(* IEC 61131-3 sources: UniTest/iecUnitTest_br/Global, 102 files *)

(* ---- Global.typ ---- *)
TYPE
    utTestCase :    STRUCT
        id : UINT; (*Identifier of the test*)
        desc : ARRAY[0..4] OF STRING[255]; (*Description of the test case*)
        state : utTestCaseStates; (*State of the test*)
        msg : STRING[255]; (*Result of the test*)
    END_STRUCT;
    utTestCaseStates :
    (
        SETUP := 0, (**)
        RUNNING := 1, (**)
        PASSED := 2, (**)
        FAILED := 3, (**)
    )
    utTestCaseSummary :    STRUCT
        Id : UINT; (*Id of the test object. Must be unique number*)
        Name : STRING[250]; (*Name of the test object*)
        TotalTests : UINT; (*Total number of tests existing*)
        TestsPassed : UINT; (*Number of tests passed*)
        TestsFailed : UINT; (*Number of tests failed*)
        PassRate : REAL; (*Pass rate % of the tests*)
        TestsRunning : BOOL; (*One or more tests are running*)
        Error : utErrors; (*Error code if error occured*)
    END_STRUCT;
    utErrors :
    (
        NO_ERROR := 0, (**)
        NO_TEST_CASES_DEFINED := 100, (**)
    )
END_TYPE

(* ---- assertArrayEqual_BYTE.st ---- *)
FUNCTION assertArrayEqual_BYTE
    (*https://github.com/tkucic/iecUnitTest/blob/main/docs/docs/ns/Global/fc/assertArrayEqual_BYTE.md*)
    vStop := (size / SIZEOF(act^[0])) - 1;

    FOR i:=0 TO vStop DO
    	pt1 := ADR(act^[i]);
    	pt2 := ADR(xp^[i]);
    	IF pt1^ <> pt2^ THEN
    		assertArrayEqual_BYTE := FALSE;
    		RETURN;
    	END_IF
    END_FOR
    (*If we reach here, all elements are equal*)
    assertArrayEqual_BYTE := TRUE;
    RETURN;

END_FUNCTION

(* ---- assertArrayEqual_DINT.st ---- *)
FUNCTION assertArrayEqual_DINT
    (*https://github.com/tkucic/iecUnitTest/blob/main/docs/docs/ns/Global/fc/assertArrayEqual_DINT.md*)
    vStop := (size / SIZEOF(act^[0])) - 1;

    FOR i:=0 TO vStop DO
    	pt1 := ADR(act^[i]);
    	pt2 := ADR(xp^[i]);
    	IF pt1^ <> pt2^ THEN
    		assertArrayEqual_DINT := FALSE;
    		RETURN;
    	END_IF
    END_FOR
    (*If we reach here, all elements are equal*)
    assertArrayEqual_DINT := TRUE;
    RETURN;

END_FUNCTION

(* ---- assertArrayEqual_DWORD.st ---- *)
FUNCTION assertArrayEqual_DWORD
    (*https://github.com/tkucic/iecUnitTest/blob/main/docs/docs/ns/Global/fc/assertArrayEqual_DWORD.md*)
    vStop := (size / SIZEOF(act^[0])) - 1;

    FOR i:=0 TO vStop DO
    	pt1 := ADR(act^[i]);
    	pt2 := ADR(xp^[i]);
    	IF pt1^ <> pt2^ THEN
    		assertArrayEqual_DWORD := FALSE;
    		RETURN;
    	END_IF
    END_FOR
    (*If we reach here, all elements are equal*)
    assertArrayEqual_DWORD := TRUE;
    RETURN;

END_FUNCTION

(* ---- assertArrayEqual_INT.st ---- *)
FUNCTION assertArrayEqual_INT
    (*https://github.com/tkucic/iecUnitTest/blob/main/docs/docs/ns/Global/fc/assertArrayEqual_INT.md*)
    vStop := (size / SIZEOF(act^[0])) - 1;

    FOR i:=0 TO vStop DO
    	pt1 := ADR(act^[i]);
    	pt2 := ADR(xp^[i]);
    	IF pt1^ <> pt2^ THEN
    		assertArrayEqual_INT := FALSE;
    		RETURN;
    	END_IF
    END_FOR
    (*If we reach here, all elements are equal*)
    assertArrayEqual_INT := TRUE;
    RETURN;

END_FUNCTION

(* ---- assertArrayEqual_LDATE.st ---- *)
FUNCTION assertArrayEqual_LDATE
    (*https://github.com/tkucic/iecUnitTest/blob/main/docs/docs/ns/Global/fc/assertArrayEqual_LDATE.md*)
    vStop := (size / SIZEOF(act^[0])) - 1;

    FOR i:=0 TO vStop DO
    	pt1 := ADR(act^[i]);
    	pt2 := ADR(xp^[i]);
    	IF pt1^ <> pt2^ THEN
    		assertArrayEqual_LDATE := FALSE;
    		RETURN;
    	END_IF
    END_FOR
    (*If we reach here, all elements are equal*)
    assertArrayEqual_LDATE := TRUE;
    RETURN;

END_FUNCTION

(* ---- assertArrayEqual_LINT.st ---- *)
FUNCTION assertArrayEqual_LINT
    (*https://github.com/tkucic/iecUnitTest/blob/main/docs/docs/ns/Global/fc/assertArrayEqual_LINT.md*)
    vStop := (size / SIZEOF(act^[0])) - 1;

    FOR i:=0 TO vStop DO
    	pt1 := ADR(act^[i]);
    	pt2 := ADR(xp^[i]);
    	IF pt1^ <> pt2^ THEN
    		assertArrayEqual_LINT := FALSE;
    		RETURN;
    	END_IF
    END_FOR
    (*If we reach here, all elements are equal*)
    assertArrayEqual_LINT := TRUE;
    RETURN;

END_FUNCTION

(* ---- assertArrayEqual_LREAL.st ---- *)
FUNCTION assertArrayEqual_LREAL
    (*https://github.com/tkucic/iecUnitTest/blob/main/docs/docs/ns/Global/fc/assertArrayEqual_LREAL.md*)
    vStop := (size / SIZEOF(act^[0])) - 1;

    FOR i:=0 TO vStop DO
    	pt1 := ADR(act^[i]);
    	pt2 := ADR(xp^[i]);
    	IF pt1^ <> pt2^ THEN
    		assertArrayEqual_LREAL := FALSE;
    		RETURN;
    	END_IF
    END_FOR
    (*If we reach here, all elements are equal*)
    assertArrayEqual_LREAL := TRUE;
    RETURN;

END_FUNCTION

(* ---- assertArrayEqual_LTIME_OF_DAY.st ---- *)
FUNCTION assertArrayEqual_LTIME_OF_DAY
    (*https://github.com/tkucic/iecUnitTest/blob/main/docs/docs/ns/Global/fc/assertArrayEqual_LTIME_OF_DAY.md*)
    vStop := (size / SIZEOF(act^[0])) - 1;

    FOR i:=0 TO vStop DO
    	pt1 := ADR(act^[i]);
    	pt2 := ADR(xp^[i]);
    	IF pt1^ <> pt2^ THEN
    		assertArrayEqual_LTIME_OF_DAY := FALSE;
    		RETURN;
    	END_IF
    END_FOR
    (*If we reach here, all elements are equal*)
    assertArrayEqual_LTIME_OF_DAY := TRUE;
    RETURN;

END_FUNCTION

(* ---- assertArrayEqual_LWORD.st ---- *)
FUNCTION assertArrayEqual_LWORD
    (*https://github.com/tkucic/iecUnitTest/blob/main/docs/docs/ns/Global/fc/assertArrayEqual_LWORD.md*)
    vStop := (size / SIZEOF(act^[0])) - 1;

    FOR i:=0 TO vStop DO
    	pt1 := ADR(act^[i]);
    	pt2 := ADR(xp^[i]);
    	IF pt1^ <> pt2^ THEN
    		assertArrayEqual_LWORD := FALSE;
    		RETURN;
    	END_IF
    END_FOR
    (*If we reach here, all elements are equal*)
    assertArrayEqual_LWORD := TRUE;
    RETURN;

END_FUNCTION

(* ---- assertArrayEqual_SINT.st ---- *)
FUNCTION assertArrayEqual_SINT
    (*https://github.com/tkucic/iecUnitTest/blob/main/docs/docs/ns/Global/fc/assertArrayEqual_SINT.md*)
    vStop := (size / SIZEOF(act^[0])) - 1;

    FOR i:=0 TO vStop DO
    	pt1 := ADR(act^[i]);
    	pt2 := ADR(xp^[i]);
    	IF pt1^ <> pt2^ THEN
    		assertArrayEqual_SINT := FALSE;
    		RETURN;
    	END_IF
    END_FOR
    (*If we reach here, all elements are equal*)
    assertArrayEqual_SINT := TRUE;
    RETURN;

END_FUNCTION

(* ---- assertArrayEqual_STRING.st ---- *)
FUNCTION assertArrayEqual_STRING
    (*https://github.com/tkucic/iecUnitTest/blob/main/docs/docs/ns/Global/fc/assertArrayEqual_STRING.md*)
    vStop := (size / SIZEOF(act^[0])) - 1;

    FOR i:=0 TO vStop DO
    	pt1 := ADR(act^[i]);
    	pt2 := ADR(xp^[i]);
    	IF pt1^ <> pt2^ THEN
    		assertArrayEqual_STRING := FALSE;
    		RETURN;
    	END_IF
    END_FOR
    (*If we reach here, all elements are equal*)
    assertArrayEqual_STRING := TRUE;
    RETURN;

END_FUNCTION

(* ---- assertArrayEqual_TIME.st ---- *)
FUNCTION assertArrayEqual_TIME
    (*https://github.com/tkucic/iecUnitTest/blob/main/docs/docs/ns/Global/fc/assertArrayEqual_TIME.md*)
    vStop := (size / SIZEOF(act^[0])) - 1;

    FOR i:=0 TO vStop DO
    	pt1 := ADR(act^[i]);
    	pt2 := ADR(xp^[i]);
    	IF pt1^ <> pt2^ THEN
    		assertArrayEqual_TIME := FALSE;
    		RETURN;
    	END_IF
    END_FOR
    (*If we reach here, all elements are equal*)
    assertArrayEqual_TIME := TRUE;
    RETURN;

END_FUNCTION

(* ---- assertArrayEqual_UDINT.st ---- *)
FUNCTION assertArrayEqual_UDINT
    (*https://github.com/tkucic/iecUnitTest/blob/main/docs/docs/ns/Global/fc/assertArrayEqual_UDINT.md*)
    vStop := (size / SIZEOF(act^[0])) - 1;

    FOR i:=0 TO vStop DO
    	pt1 := ADR(act^[i]);
    	pt2 := ADR(xp^[i]);
    	IF pt1^ <> pt2^ THEN
    		assertArrayEqual_UDINT := FALSE;
    		RETURN;
    	END_IF
    END_FOR
    (*If we reach here, all elements are equal*)
    assertArrayEqual_UDINT := TRUE;
    RETURN;

END_FUNCTION

(* ---- assertArrayEqual_UINT.st ---- *)
FUNCTION assertArrayEqual_UINT
    (*https://github.com/tkucic/iecUnitTest/blob/main/docs/docs/ns/Global/fc/assertArrayEqual_UINT.md*)
    vStop := (size / SIZEOF(act^[0])) - 1;

    FOR i:=0 TO vStop DO
    	pt1 := ADR(act^[i]);
    	pt2 := ADR(xp^[i]);
    	IF pt1^ <> pt2^ THEN
    		assertArrayEqual_UINT := FALSE;
    		RETURN;
    	END_IF
    END_FOR
    (*If we reach here, all elements are equal*)
    assertArrayEqual_UINT := TRUE;
    RETURN;

END_FUNCTION

(* ---- assertArrayEqual_ULINT.st ---- *)
FUNCTION assertArrayEqual_ULINT
    (*https://github.com/tkucic/iecUnitTest/blob/main/docs/docs/ns/Global/fc/assertArrayEqual_ULINT.md*)
    vStop := (size / SIZEOF(act^[0])) - 1;

    FOR i:=0 TO vStop DO
    	pt1 := ADR(act^[i]);
    	pt2 := ADR(xp^[i]);
    	IF pt1^ <> pt2^ THEN
    		assertArrayEqual_ULINT := FALSE;
    		RETURN;
    	END_IF
    END_FOR
    (*If we reach here, all elements are equal*)
    assertArrayEqual_ULINT := TRUE;
    RETURN;

END_FUNCTION

(* ---- assertArrayEqual_WORD.st ---- *)
FUNCTION assertArrayEqual_WORD
    (*https://github.com/tkucic/iecUnitTest/blob/main/docs/docs/ns/Global/fc/assertArrayEqual_WORD.md*)
    vStop := (size / SIZEOF(act^[0])) - 1;

    FOR i:=0 TO vStop DO
    	pt1 := ADR(act^[i]);
    	pt2 := ADR(xp^[i]);
    	IF pt1^ <> pt2^ THEN
    		assertArrayEqual_WORD := FALSE;
    		RETURN;
    	END_IF
    END_FOR
    (*If we reach here, all elements are equal*)
    assertArrayEqual_WORD := TRUE;
    RETURN;

END_FUNCTION

(* ---- assertArrayEqual_WSTRING.st ---- *)
FUNCTION assertArrayEqual_WSTRING
    (*https://github.com/tkucic/iecUnitTest/blob/main/docs/docs/ns/Global/fc/assertArrayEqual_WSTRING.md*)
    vStop := (size / SIZEOF(act^[0])) - 1;

    FOR i:=0 TO vStop DO
    	pt1 := ADR(act^[i]);
    	pt2 := ADR(xp^[i]);
    	IF pt1^ <> pt2^ THEN
    		assertArrayEqual_WSTRING := FALSE;
    		RETURN;
    	END_IF
    END_FOR
    (*If we reach here, all elements are equal*)
    assertArrayEqual_WSTRING := TRUE;
    RETURN;

END_FUNCTION

(* ---- assertEqual_BYTE.st ---- *)
FUNCTION assertEqual_BYTE
    (*https://github.com/tkucic/iecUnitTest/blob/main/docs/docs/ns/Global/fc/assertEqual_BYTE.md*)
    assertEqual_BYTE := act = xp;
    RETURN;

END_FUNCTION

(* ---- assertEqual_DATE_AND_TIME.st ---- *)
FUNCTION assertEqual_DATE_AND_TIME
    (*https://github.com/tkucic/iecUnitTest/blob/main/docs/docs/ns/Global/fc/assertEqual_DATE_AND_TIME.md*)
    assertEqual_DATE_AND_TIME := act = xp;
    RETURN;

END_FUNCTION

(* ---- assertEqual_DWORD.st ---- *)
FUNCTION assertEqual_DWORD
    (*https://github.com/tkucic/iecUnitTest/blob/main/docs/docs/ns/Global/fc/assertEqual_DWORD.md*)
    assertEqual_DWORD := act = xp;
    RETURN;

END_FUNCTION

(* ---- assertEqual_INT.st ---- *)
FUNCTION assertEqual_INT
    (*https://github.com/tkucic/iecUnitTest/blob/main/docs/docs/ns/Global/fc/assertEqual_INT.md*)
    assertEqual_INT := act = xp;
    RETURN;

END_FUNCTION

(* ---- assertEqual_LDATE.st ---- *)
FUNCTION assertEqual_LDATE
    (*https://github.com/tkucic/iecUnitTest/blob/main/docs/docs/ns/Global/fc/assertEqual_LDATE.md*)
    assertEqual_LDATE := act = xp;
    RETURN;

END_FUNCTION

(* ---- assertEqual_LDATE_AND_TIME.st ---- *)
FUNCTION assertEqual_LDATE_AND_TIME
    (*https://github.com/tkucic/iecUnitTest/blob/main/docs/docs/ns/Global/fc/assertEqual_LDATE_AND_TIME.md*)
    assertEqual_LDATE_AND_TIME := act = xp;
    RETURN;

END_FUNCTION

(* ---- assertEqual_LINT.st ---- *)
FUNCTION assertEqual_LINT
    (*https://github.com/tkucic/iecUnitTest/blob/main/docs/docs/ns/Global/fc/assertEqual_LINT.md*)
    assertEqual_LINT := act = xp;
    RETURN;

END_FUNCTION

(* ---- assertEqual_LTIME.st ---- *)
FUNCTION assertEqual_LTIME
    (*https://github.com/tkucic/iecUnitTest/blob/main/docs/docs/ns/Global/fc/assertEqual_LTIME.md*)
    assertEqual_LTIME := act = xp;
    RETURN;

END_FUNCTION

(* ---- assertEqual_LTIME_OF_DAY.st ---- *)
FUNCTION assertEqual_LTIME_OF_DAY
    (*https://github.com/tkucic/iecUnitTest/blob/main/docs/docs/ns/Global/fc/assertEqual_LTIME_OF_DAY.md*)
    assertEqual_LTIME_OF_DAY := act = xp;
    RETURN;

END_FUNCTION

(* ---- assertEqual_REAL.st ---- *)
FUNCTION assertEqual_REAL
    (*https://github.com/tkucic/iecUnitTest/blob/main/docs/docs/ns/Global/fc/assertEqual_REAL.md*)
    assertEqual_REAL := act = xp;
    RETURN;

END_FUNCTION

(* ---- assertEqual_STRING.st ---- *)
FUNCTION assertEqual_STRING
    (*https://github.com/tkucic/iecUnitTest/blob/main/docs/docs/ns/Global/fc/assertEqual_STRING.md*)
    assertEqual_STRING := act = xp;
    RETURN;

END_FUNCTION

(* ---- assertEqual_UDINT.st ---- *)
FUNCTION assertEqual_UDINT
    (*https://github.com/tkucic/iecUnitTest/blob/main/docs/docs/ns/Global/fc/assertEqual_UDINT.md*)
    assertEqual_UDINT := act = xp;
    RETURN;

END_FUNCTION

(* ---- assertEqual_ULINT.st ---- *)
FUNCTION assertEqual_ULINT
    (*https://github.com/tkucic/iecUnitTest/blob/main/docs/docs/ns/Global/fc/assertEqual_ULINT.md*)
    assertEqual_ULINT := act = xp;
    RETURN;

END_FUNCTION

(* ---- assertEqual_USINT.st ---- *)
FUNCTION assertEqual_USINT
    (*https://github.com/tkucic/iecUnitTest/blob/main/docs/docs/ns/Global/fc/assertEqual_USINT.md*)
    assertEqual_USINT := act = xp;
    RETURN;

END_FUNCTION

(* ---- assertFalse.st ---- *)
FUNCTION assertFalse
    (*https://github.com/tkucic/iecUnitTest/blob/main/docs/docs/ns/Global/fc/assertFalse.md*)
    assertFalse := NOT condition;
    RETURN;

END_FUNCTION

(* ---- assertGreater_BYTE.st ---- *)
FUNCTION assertGreater_BYTE
    (*https://github.com/tkucic/iecUnitTest/blob/main/docs/docs/ns/Global/fc/assertGreater_BYTE.md*)
    assertGreater_BYTE := act > xp;
    RETURN;

END_FUNCTION

(* ---- assertGreater_DATE.st ---- *)
FUNCTION assertGreater_DATE
    (*https://github.com/tkucic/iecUnitTest/blob/main/docs/docs/ns/Global/fc/assertGreater_DATE.md*)
    assertGreater_DATE := act > xp;
    RETURN;

END_FUNCTION

(* ---- assertGreater_DWORD.st ---- *)
FUNCTION assertGreater_DWORD
    (*https://github.com/tkucic/iecUnitTest/blob/main/docs/docs/ns/Global/fc/assertGreater_DWORD.md*)
    assertGreater_DWORD := act > xp;
    RETURN;

END_FUNCTION

(* ---- assertGreater_INT.st ---- *)
FUNCTION assertGreater_INT
    (*https://github.com/tkucic/iecUnitTest/blob/main/docs/docs/ns/Global/fc/assertGreater_INT.md*)
    assertGreater_INT := act > xp;
    RETURN;

END_FUNCTION

(* ---- assertGreater_LDATE_AND_TIME.st ---- *)
FUNCTION assertGreater_LDATE_AND_TIME
    (*https://github.com/tkucic/iecUnitTest/blob/main/docs/docs/ns/Global/fc/assertGreater_LDATE_AND_TIME.md*)
    assertGreater_LDATE_AND_TIME := act > xp;
    RETURN;

END_FUNCTION

(* ---- assertGreater_LREAL.st ---- *)
FUNCTION assertGreater_LREAL
    (*https://github.com/tkucic/iecUnitTest/blob/main/docs/docs/ns/Global/fc/assertGreater_LREAL.md*)
    assertGreater_LREAL := act > xp;
    RETURN;

END_FUNCTION

(* ---- assertGreater_LTIME.st ---- *)
FUNCTION assertGreater_LTIME
    (*https://github.com/tkucic/iecUnitTest/blob/main/docs/docs/ns/Global/fc/assertGreater_LTIME.md*)
    assertGreater_LTIME := act > xp;
    RETURN;

END_FUNCTION

(* ---- assertGreater_LTIME_OF_DAY.st ---- *)
FUNCTION assertGreater_LTIME_OF_DAY
    (*https://github.com/tkucic/iecUnitTest/blob/main/docs/docs/ns/Global/fc/assertGreater_LTIME_OF_DAY.md*)
    assertGreater_LTIME_OF_DAY := act > xp;
    RETURN;

END_FUNCTION

(* ---- assertGreater_LWORD.st ---- *)
FUNCTION assertGreater_LWORD
    (*https://github.com/tkucic/iecUnitTest/blob/main/docs/docs/ns/Global/fc/assertGreater_LWORD.md*)
    assertGreater_LWORD := act > xp;
    RETURN;

END_FUNCTION

(* ---- assertGreater_REAL.st ---- *)
FUNCTION assertGreater_REAL
    (*https://github.com/tkucic/iecUnitTest/blob/main/docs/docs/ns/Global/fc/assertGreater_REAL.md*)
    assertGreater_REAL := act > xp;
    RETURN;

END_FUNCTION

(* ---- assertGreater_SINT.st ---- *)
FUNCTION assertGreater_SINT
    (*https://github.com/tkucic/iecUnitTest/blob/main/docs/docs/ns/Global/fc/assertGreater_SINT.md*)
    assertGreater_SINT := act > xp;
    RETURN;

END_FUNCTION

(* ---- assertGreater_TIME.st ---- *)
FUNCTION assertGreater_TIME
    (*https://github.com/tkucic/iecUnitTest/blob/main/docs/docs/ns/Global/fc/assertGreater_TIME.md*)
    assertGreater_TIME := act > xp;
    RETURN;

END_FUNCTION

(* ---- assertGreater_TIME_OF_DAY.st ---- *)
FUNCTION assertGreater_TIME_OF_DAY
    (*https://github.com/tkucic/iecUnitTest/blob/main/docs/docs/ns/Global/fc/assertGreater_TIME_OF_DAY.md*)
    assertGreater_TIME_OF_DAY := act > xp;
    RETURN;

END_FUNCTION

(* ---- assertGreater_UINT.st ---- *)
FUNCTION assertGreater_UINT
    (*https://github.com/tkucic/iecUnitTest/blob/main/docs/docs/ns/Global/fc/assertGreater_UINT.md*)
    assertGreater_UINT := act > xp;
    RETURN;

END_FUNCTION

(* ---- assertGreater_ULINT.st ---- *)
FUNCTION assertGreater_ULINT
    (*https://github.com/tkucic/iecUnitTest/blob/main/docs/docs/ns/Global/fc/assertGreater_ULINT.md*)
    assertGreater_ULINT := act > xp;
    RETURN;

END_FUNCTION

(* ---- assertGreater_WORD.st ---- *)
FUNCTION assertGreater_WORD
    (*https://github.com/tkucic/iecUnitTest/blob/main/docs/docs/ns/Global/fc/assertGreater_WORD.md*)
    assertGreater_WORD := act > xp;
    RETURN;

END_FUNCTION

(* ---- assertGreaterEqual_BYTE.st ---- *)
FUNCTION assertGreaterEqual_BYTE
    (*https://github.com/tkucic/iecUnitTest/blob/main/docs/docs/ns/Global/fc/assertGreaterEqual_BYTE.md*)
    assertGreaterEqual_BYTE := act >= xp;
    RETURN;

END_FUNCTION

(* ---- assertGreaterEqual_DWORD.st ---- *)
FUNCTION assertGreaterEqual_DWORD
    (*https://github.com/tkucic/iecUnitTest/blob/main/docs/docs/ns/Global/fc/assertGreaterEqual_DWORD.md*)
    assertGreaterEqual_DWORD := act >= xp;
    RETURN;

END_FUNCTION

(* ---- assertGreaterEqual_LDATE_AND_TIME.st ---- *)
FUNCTION assertGreaterEqual_LDATE_AND_TIME
    (*https://github.com/tkucic/iecUnitTest/blob/main/docs/docs/ns/Global/fc/assertGreaterEqual_LDATE_AND_TIME.md*)
    assertGreaterEqual_LDATE_AND_TIME := act >= xp;
    RETURN;

END_FUNCTION

(* ---- assertGreaterEqual_LTIME_OF_DAY.st ---- *)
FUNCTION assertGreaterEqual_LTIME_OF_DAY
    (*https://github.com/tkucic/iecUnitTest/blob/main/docs/docs/ns/Global/fc/assertGreaterEqual_LTIME_OF_DAY.md*)
    assertGreaterEqual_LTIME_OF_DAY := act >= xp;
    RETURN;

END_FUNCTION

(* ---- assertGreaterEqual_LWORD.st ---- *)
FUNCTION assertGreaterEqual_LWORD
    (*https://github.com/tkucic/iecUnitTest/blob/main/docs/docs/ns/Global/fc/assertGreaterEqual_LWORD.md*)
    assertGreaterEqual_LWORD := act >= xp;
    RETURN;

END_FUNCTION

(* ---- assertGreaterEqual_SINT.st ---- *)
FUNCTION assertGreaterEqual_SINT
    (*https://github.com/tkucic/iecUnitTest/blob/main/docs/docs/ns/Global/fc/assertGreaterEqual_SINT.md*)
    assertGreaterEqual_SINT := act >= xp;
    RETURN;

END_FUNCTION

(* ---- assertGreaterEqual_TIME_OF_DAY.st ---- *)
FUNCTION assertGreaterEqual_TIME_OF_DAY
    (*https://github.com/tkucic/iecUnitTest/blob/main/docs/docs/ns/Global/fc/assertGreaterEqual_TIME_OF_DAY.md*)
    assertGreaterEqual_TIME_OF_DAY := act >= xp;
    RETURN;

END_FUNCTION

(* ---- assertGreaterEqual_UDINT.st ---- *)
FUNCTION assertGreaterEqual_UDINT
    (*https://github.com/tkucic/iecUnitTest/blob/main/docs/docs/ns/Global/fc/assertGreaterEqual_UDINT.md*)
    assertGreaterEqual_UDINT := act >= xp;
    RETURN;

END_FUNCTION

(* ---- assertGreaterEqual_UINT.st ---- *)
FUNCTION assertGreaterEqual_UINT
    (*https://github.com/tkucic/iecUnitTest/blob/main/docs/docs/ns/Global/fc/assertGreaterEqual_UINT.md*)
    assertGreaterEqual_UINT := act >= xp;
    RETURN;

END_FUNCTION

(* ---- assertGreaterEqual_ULINT.st ---- *)
FUNCTION assertGreaterEqual_ULINT
    (*https://github.com/tkucic/iecUnitTest/blob/main/docs/docs/ns/Global/fc/assertGreaterEqual_ULINT.md*)
    assertGreaterEqual_ULINT := act >= xp;
    RETURN;

END_FUNCTION

(* ---- assertGreaterEqual_USINT.st ---- *)
FUNCTION assertGreaterEqual_USINT
    (*https://github.com/tkucic/iecUnitTest/blob/main/docs/docs/ns/Global/fc/assertGreaterEqual_USINT.md*)
    assertGreaterEqual_USINT := act >= xp;
    RETURN;

END_FUNCTION

(* ---- assertLess_DATE_AND_TIME.st ---- *)
FUNCTION assertLess_DATE_AND_TIME
    (*https://github.com/tkucic/iecUnitTest/blob/main/docs/docs/ns/Global/fc/assertLess_DATE_AND_TIME.md*)
    assertLess_DATE_AND_TIME := act < xp;
    RETURN;

END_FUNCTION

(* ---- assertLess_DWORD.st ---- *)
FUNCTION assertLess_DWORD
    (*https://github.com/tkucic/iecUnitTest/blob/main/docs/docs/ns/Global/fc/assertLess_DWORD.md*)
    assertLess_DWORD := act < xp;
    RETURN;

END_FUNCTION

(* ---- assertLess_INT.st ---- *)
FUNCTION assertLess_INT
    (*https://github.com/tkucic/iecUnitTest/blob/main/docs/docs/ns/Global/fc/assertLess_INT.md*)
    assertLess_INT := act < xp;
    RETURN;

END_FUNCTION

(* ---- assertLess_LINT.st ---- *)
FUNCTION assertLess_LINT
    (*https://github.com/tkucic/iecUnitTest/blob/main/docs/docs/ns/Global/fc/assertLess_LINT.md*)
    assertLess_LINT := act < xp;
    RETURN;

END_FUNCTION

(* ---- assertLess_LTIME.st ---- *)
FUNCTION assertLess_LTIME
    (*https://github.com/tkucic/iecUnitTest/blob/main/docs/docs/ns/Global/fc/assertLess_LTIME.md*)
    assertLess_LTIME := act < xp;
    RETURN;

END_FUNCTION

(* ---- assertLess_LTIME_OF_DAY.st ---- *)
FUNCTION assertLess_LTIME_OF_DAY
    (*https://github.com/tkucic/iecUnitTest/blob/main/docs/docs/ns/Global/fc/assertLess_LTIME_OF_DAY.md*)
    assertLess_LTIME_OF_DAY := act < xp;
    RETURN;

END_FUNCTION

(* ---- assertLess_LWORD.st ---- *)
FUNCTION assertLess_LWORD
    (*https://github.com/tkucic/iecUnitTest/blob/main/docs/docs/ns/Global/fc/assertLess_LWORD.md*)
    assertLess_LWORD := act < xp;
    RETURN;

END_FUNCTION

(* ---- assertLess_SINT.st ---- *)
FUNCTION assertLess_SINT
    (*https://github.com/tkucic/iecUnitTest/blob/main/docs/docs/ns/Global/fc/assertLess_SINT.md*)
    assertLess_SINT := act < xp;
    RETURN;

END_FUNCTION

(* ---- assertLess_TIME.st ---- *)
FUNCTION assertLess_TIME
    (*https://github.com/tkucic/iecUnitTest/blob/main/docs/docs/ns/Global/fc/assertLess_TIME.md*)
    assertLess_TIME := act < xp;
    RETURN;

END_FUNCTION

(* ---- assertLess_TIME_OF_DAY.st ---- *)
FUNCTION assertLess_TIME_OF_DAY
    (*https://github.com/tkucic/iecUnitTest/blob/main/docs/docs/ns/Global/fc/assertLess_TIME_OF_DAY.md*)
    assertLess_TIME_OF_DAY := act < xp;
    RETURN;

END_FUNCTION

(* ---- assertLess_UDINT.st ---- *)
FUNCTION assertLess_UDINT
    (*https://github.com/tkucic/iecUnitTest/blob/main/docs/docs/ns/Global/fc/assertLess_UDINT.md*)
    assertLess_UDINT := act < xp;
    RETURN;

END_FUNCTION

(* ---- assertLess_USINT.st ---- *)
FUNCTION assertLess_USINT
    (*https://github.com/tkucic/iecUnitTest/blob/main/docs/docs/ns/Global/fc/assertLess_USINT.md*)
    assertLess_USINT := act < xp;
    RETURN;

END_FUNCTION

(* ---- assertLess_WORD.st ---- *)
FUNCTION assertLess_WORD
    (*https://github.com/tkucic/iecUnitTest/blob/main/docs/docs/ns/Global/fc/assertLess_WORD.md*)
    assertLess_WORD := act < xp;
    RETURN;

END_FUNCTION

(* ---- assertLessEqual_BYTE.st ---- *)
FUNCTION assertLessEqual_BYTE
    (*https://github.com/tkucic/iecUnitTest/blob/main/docs/docs/ns/Global/fc/assertLessEqual_BYTE.md*)
    assertLessEqual_BYTE := act <= xp;
    RETURN;

END_FUNCTION

(* ---- assertLessEqual_DATE.st ---- *)
FUNCTION assertLessEqual_DATE
    (*https://github.com/tkucic/iecUnitTest/blob/main/docs/docs/ns/Global/fc/assertLessEqual_DATE.md*)
    assertLessEqual_DATE := act <= xp;
    RETURN;

END_FUNCTION

(* ---- assertLessEqual_DINT.st ---- *)
FUNCTION assertLessEqual_DINT
    (*https://github.com/tkucic/iecUnitTest/blob/main/docs/docs/ns/Global/fc/assertLessEqual_DINT.md*)
    assertLessEqual_DINT := act <= xp;
    RETURN;

END_FUNCTION

(* ---- assertLessEqual_LDATE.st ---- *)
FUNCTION assertLessEqual_LDATE
    (*https://github.com/tkucic/iecUnitTest/blob/main/docs/docs/ns/Global/fc/assertLessEqual_LDATE.md*)
    assertLessEqual_LDATE := act <= xp;
    RETURN;

END_FUNCTION

(* ---- assertLessEqual_LDATE_AND_TIME.st ---- *)
FUNCTION assertLessEqual_LDATE_AND_TIME
    (*https://github.com/tkucic/iecUnitTest/blob/main/docs/docs/ns/Global/fc/assertLessEqual_LDATE_AND_TIME.md*)
    assertLessEqual_LDATE_AND_TIME := act <= xp;
    RETURN;

END_FUNCTION

(* ---- assertLessEqual_LREAL.st ---- *)
FUNCTION assertLessEqual_LREAL
    (*https://github.com/tkucic/iecUnitTest/blob/main/docs/docs/ns/Global/fc/assertLessEqual_LREAL.md*)
    assertLessEqual_LREAL := act <= xp;
    RETURN;

END_FUNCTION

(* ---- assertLessEqual_LTIME.st ---- *)
FUNCTION assertLessEqual_LTIME
    (*https://github.com/tkucic/iecUnitTest/blob/main/docs/docs/ns/Global/fc/assertLessEqual_LTIME.md*)
    assertLessEqual_LTIME := act <= xp;
    RETURN;

END_FUNCTION

(* ---- assertLessEqual_LTIME_OF_DAY.st ---- *)
FUNCTION assertLessEqual_LTIME_OF_DAY
    (*https://github.com/tkucic/iecUnitTest/blob/main/docs/docs/ns/Global/fc/assertLessEqual_LTIME_OF_DAY.md*)
    assertLessEqual_LTIME_OF_DAY := act <= xp;
    RETURN;

END_FUNCTION

(* ---- assertLessEqual_REAL.st ---- *)
FUNCTION assertLessEqual_REAL
    (*https://github.com/tkucic/iecUnitTest/blob/main/docs/docs/ns/Global/fc/assertLessEqual_REAL.md*)
    assertLessEqual_REAL := act <= xp;
    RETURN;

END_FUNCTION

(* ---- assertLessEqual_TIME.st ---- *)
FUNCTION assertLessEqual_TIME
    (*https://github.com/tkucic/iecUnitTest/blob/main/docs/docs/ns/Global/fc/assertLessEqual_TIME.md*)
    assertLessEqual_TIME := act <= xp;
    RETURN;

END_FUNCTION

(* ---- assertLessEqual_UDINT.st ---- *)
FUNCTION assertLessEqual_UDINT
    (*https://github.com/tkucic/iecUnitTest/blob/main/docs/docs/ns/Global/fc/assertLessEqual_UDINT.md*)
    assertLessEqual_UDINT := act <= xp;
    RETURN;

END_FUNCTION

(* ---- assertLessEqual_UINT.st ---- *)
FUNCTION assertLessEqual_UINT
    (*https://github.com/tkucic/iecUnitTest/blob/main/docs/docs/ns/Global/fc/assertLessEqual_UINT.md*)
    assertLessEqual_UINT := act <= xp;
    RETURN;

END_FUNCTION

(* ---- assertLessEqual_ULINT.st ---- *)
FUNCTION assertLessEqual_ULINT
    (*https://github.com/tkucic/iecUnitTest/blob/main/docs/docs/ns/Global/fc/assertLessEqual_ULINT.md*)
    assertLessEqual_ULINT := act <= xp;
    RETURN;

END_FUNCTION

(* ---- assertLessEqual_USINT.st ---- *)
FUNCTION assertLessEqual_USINT
    (*https://github.com/tkucic/iecUnitTest/blob/main/docs/docs/ns/Global/fc/assertLessEqual_USINT.md*)
    assertLessEqual_USINT := act <= xp;
    RETURN;

END_FUNCTION

(* ---- assertLessEqual_WORD.st ---- *)
FUNCTION assertLessEqual_WORD
    (*https://github.com/tkucic/iecUnitTest/blob/main/docs/docs/ns/Global/fc/assertLessEqual_WORD.md*)
    assertLessEqual_WORD := act <= xp;
    RETURN;

END_FUNCTION

(* ---- assertNotEqual_BYTE.st ---- *)
FUNCTION assertNotEqual_BYTE
    (*https://github.com/tkucic/iecUnitTest/blob/main/docs/docs/ns/Global/fc/assertNotEqual_BYTE.md*)
    assertNotEqual_BYTE := act <> xp;
    RETURN;

END_FUNCTION

(* ---- assertNotEqual_DATE.st ---- *)
FUNCTION assertNotEqual_DATE
    (*https://github.com/tkucic/iecUnitTest/blob/main/docs/docs/ns/Global/fc/assertNotEqual_DATE.md*)
    assertNotEqual_DATE := act <> xp;
    RETURN;

END_FUNCTION

(* ---- assertNotEqual_INT.st ---- *)
FUNCTION assertNotEqual_INT
    (*https://github.com/tkucic/iecUnitTest/blob/main/docs/docs/ns/Global/fc/assertNotEqual_INT.md*)
    assertNotEqual_INT := act <> xp;
    RETURN;

END_FUNCTION

(* ---- assertNotEqual_LDATE_AND_TIME.st ---- *)
FUNCTION assertNotEqual_LDATE_AND_TIME
    (*https://github.com/tkucic/iecUnitTest/blob/main/docs/docs/ns/Global/fc/assertNotEqual_LDATE_AND_TIME.md*)
    assertNotEqual_LDATE_AND_TIME := act <> xp;
    RETURN;

END_FUNCTION

(* ---- assertNotEqual_LINT.st ---- *)
FUNCTION assertNotEqual_LINT
    (*https://github.com/tkucic/iecUnitTest/blob/main/docs/docs/ns/Global/fc/assertNotEqual_LINT.md*)
    assertNotEqual_LINT := act <> xp;
    RETURN;

END_FUNCTION

(* ---- assertNotEqual_LTIME.st ---- *)
FUNCTION assertNotEqual_LTIME
    (*https://github.com/tkucic/iecUnitTest/blob/main/docs/docs/ns/Global/fc/assertNotEqual_LTIME.md*)
    assertNotEqual_LTIME := act <> xp;
    RETURN;

END_FUNCTION

(* ---- assertNotEqual_LTIME_OF_DAY.st ---- *)
FUNCTION assertNotEqual_LTIME_OF_DAY
    (*https://github.com/tkucic/iecUnitTest/blob/main/docs/docs/ns/Global/fc/assertNotEqual_LTIME_OF_DAY.md*)
    assertNotEqual_LTIME_OF_DAY := act <> xp;
    RETURN;

END_FUNCTION

(* ---- assertNotEqual_SINT.st ---- *)
FUNCTION assertNotEqual_SINT
    (*https://github.com/tkucic/iecUnitTest/blob/main/docs/docs/ns/Global/fc/assertNotEqual_SINT.md*)
    assertNotEqual_SINT := act <> xp;
    RETURN;

END_FUNCTION

(* ---- assertNotEqual_STRING.st ---- *)
FUNCTION assertNotEqual_STRING
    (*https://github.com/tkucic/iecUnitTest/blob/main/docs/docs/ns/Global/fc/assertNotEqual_STRING.md*)
    assertNotEqual_STRING := act <> xp;
    RETURN;

END_FUNCTION

(* ---- assertNotEqual_UDINT.st ---- *)
FUNCTION assertNotEqual_UDINT
    (*https://github.com/tkucic/iecUnitTest/blob/main/docs/docs/ns/Global/fc/assertNotEqual_UDINT.md*)
    assertNotEqual_UDINT := act <> xp;
    RETURN;

END_FUNCTION

(* ---- assertNotEqual_WORD.st ---- *)
FUNCTION assertNotEqual_WORD
    (*https://github.com/tkucic/iecUnitTest/blob/main/docs/docs/ns/Global/fc/assertNotEqual_WORD.md*)
    assertNotEqual_WORD := act <> xp;
    RETURN;

END_FUNCTION

(* ---- Global.fun ---- *)
FUNCTION_BLOCK utTestSuite (* Enables running, resetting and reporting for tests cases defined of a POU under test *)(* https://github.com/tkucic/iecUnitTest/blob/main/docs/docs/ns/Global/fb/utTestSuite.md *)
    VAR_INPUT
        Id : UINT; (*Id of the test object. Must be unique number*)
        Name : STRING[250]; (*Name of the test object*)
        RunTests : BOOL; (*Starts all tests that are in setup state. Sets state to running.*)
        ResetTests : BOOL; (*Sets state to setup on test cases that are PASSED or FAILED.*)
    END_VAR
    VAR_IN_OUT
        TestCases : ARRAY[0..20] OF utTestCase; (*Array of test case definition*)
    END_VAR
    VAR_OUTPUT
        Summary : utTestCaseSummary; (*Summary of the test results*)
    END_VAR
    VAR
        i : UINT; (*Iterator variable*)
        runCmd : R_TRIG; (*Trigger to prevent constant run commands*)
        resetCmd : R_TRIG; (*Trigger to prevent constant reset commands*)
    END_VAR
END_FUNCTION_BLOCK
FUNCTION_BLOCK utTestReporter (* Provides feedback on the status of tests on a system scale *)(* https://github.com/tkucic/iecUnitTest/blob/main/docs/docs/ns/Global/fb/utTestReporter.md *)
    VAR_IN_OUT
        Results : ARRAY[0..500] OF utTestCaseSummary; (*Summaries of tests for each POU under test*)
    END_VAR
    VAR_OUTPUT
        NrPousUnderTest : UINT; (*Total number of POUs under test*)
        NrOfTests : UINT; (*Total number of tests*)
        NrTestsPassed : UINT; (*Number of tests passed*)
        NrTestsFailed : UINT; (*Number of tests failed*)
        PassRate : REAL; (*Total pass rate*)
        TestsInProgress : BOOL; (*Indicates that one or more tests are in progress*)
        Error : BOOL; (*Indicates that one or more tests are in error state*)
    END_VAR
    VAR
        i : UINT; (*Iterator variable*)
    END_VAR
END_FUNCTION_BLOCK
FUNCTION assertFalse : BOOL (* Returns TRUE if condition is NOT TRUE *)(* https://github.com/tkucic/iecUnitTest/blob/main/docs/docs/ns/Global/fc/assertFalse.md *)
    VAR_INPUT
        condition : BOOL; (*Variable to test*)
    END_VAR
END_FUNCTION
FUNCTION assertEqual_BOOL : BOOL (* Returns TRUE if act = xp. *)(* https://github.com/tkucic/iecUnitTest/blob/main/docs/docs/ns/Global/fc/assertEqual_BOOL.md *)
    VAR_INPUT
        act : BOOL; (*Variable to test*)
        xp : BOOL; (*Variable to test against*)
    END_VAR
END_FUNCTION
FUNCTION assertEqual_BYTE : BOOL (* Returns TRUE if act = xp. *)(* https://github.com/tkucic/iecUnitTest/blob/main/docs/docs/ns/Global/fc/assertEqual_BYTE.md *)
    VAR_INPUT
        act : BYTE; (*Variable to test*)
        xp : BYTE; (*Variable to test against*)
    END_VAR
END_FUNCTION
FUNCTION assertEqual_WORD : BOOL (* Returns TRUE if act = xp. *)(* https://github.com/tkucic/iecUnitTest/blob/main/docs/docs/ns/Global/fc/assertEqual_WORD.md *)
    VAR_INPUT
        act : WORD; (*Variable to test*)
        xp : WORD; (*Variable to test against*)
    END_VAR
END_FUNCTION
FUNCTION assertEqual_DWORD : BOOL (* Returns TRUE if act = xp. *)(* https://github.com/tkucic/iecUnitTest/blob/main/docs/docs/ns/Global/fc/assertEqual_DWORD.md *)
    VAR_INPUT
        act : DWORD; (*Variable to test*)
        xp : DWORD; (*Variable to test against*)
    END_VAR
END_FUNCTION
FUNCTION assertEqual_LWORD : BOOL (* Returns TRUE if act = xp. *)(* https://github.com/tkucic/iecUnitTest/blob/main/docs/docs/ns/Global/fc/assertEqual_LWORD.md *)
    VAR_INPUT
        act : LWORD; (*Variable to test*)
        xp : LWORD; (*Variable to test against*)
    END_VAR
END_FUNCTION
FUNCTION assertEqual_SINT : BOOL (* Returns TRUE if act = xp. *)(* https://github.com/tkucic/iecUnitTest/blob/main/docs/docs/ns/Global/fc/assertEqual_SINT.md *)
    VAR_INPUT
        act : SINT; (*Variable to test*)
        xp : SINT; (*Variable to test against*)
    END_VAR
END_FUNCTION
FUNCTION assertEqual_USINT : BOOL (* Returns TRUE if act = xp. *)(* https://github.com/tkucic/iecUnitTest/blob/main/docs/docs/ns/Global/fc/assertEqual_USINT.md *)
    VAR_INPUT
        act : USINT; (*Variable to test*)
        xp : USINT; (*Variable to test against*)
    END_VAR
END_FUNCTION
FUNCTION assertEqual_INT : BOOL (* Returns TRUE if act = xp. *)(* https://github.com/tkucic/iecUnitTest/blob/main/docs/docs/ns/Global/fc/assertEqual_INT.md *)
    VAR_INPUT
        act : INT; (*Variable to test*)
        xp : INT; (*Variable to test against*)
    END_VAR
END_FUNCTION
FUNCTION assertEqual_UINT : BOOL (* Returns TRUE if act = xp. *)(* https://github.com/tkucic/iecUnitTest/blob/main/docs/docs/ns/Global/fc/assertEqual_UINT.md *)
    VAR_INPUT
        act : UINT; (*Variable to test*)
        xp : UINT; (*Variable to test against*)
    END_VAR
END_FUNCTION
FUNCTION assertEqual_DINT : BOOL (* Returns TRUE if act = xp. *)(* https://github.com/tkucic/iecUnitTest/blob/main/docs/docs/ns/Global/fc/assertEqual_DINT.md *)
    VAR_INPUT
        act : DINT; (*Variable to test*)
        xp : DINT; (*Variable to test against*)
    END_VAR
END_FUNCTION
FUNCTION assertEqual_UDINT : BOOL (* Returns TRUE if act = xp. *)(* https://github.com/tkucic/iecUnitTest/blob/main/docs/docs/ns/Global/fc/assertEqual_UDINT.md *)
    VAR_INPUT
        act : UDINT; (*Variable to test*)
        xp : UDINT; (*Variable to test against*)
    END_VAR
END_FUNCTION
FUNCTION assertEqual_LINT : BOOL (* Returns TRUE if act = xp. *)(* https://github.com/tkucic/iecUnitTest/blob/main/docs/docs/ns/Global/fc/assertEqual_LINT.md *)
    VAR_INPUT
        act : LINT; (*Variable to test*)
        xp : LINT; (*Variable to test against*)
    END_VAR
END_FUNCTION
FUNCTION assertEqual_ULINT : BOOL (* Returns TRUE if act = xp. *)(* https://github.com/tkucic/iecUnitTest/blob/main/docs/docs/ns/Global/fc/assertEqual_ULINT.md *)
    VAR_INPUT
        act : ULINT; (*Variable to test*)
        xp : ULINT; (*Variable to test against*)
    END_VAR
END_FUNCTION
FUNCTION assertEqual_REAL : BOOL (* Returns TRUE if act = xp. *)(* https://github.com/tkucic/iecUnitTest/blob/main/docs/docs/ns/Global/fc/assertEqual_REAL.md *)
    VAR_INPUT
        act : REAL; (*Variable to test*)
        xp : REAL; (*Variable to test against*)
    END_VAR
END_FUNCTION
FUNCTION assertEqual_LREAL : BOOL (* Returns TRUE if act = xp. *)(* https://github.com/tkucic/iecUnitTest/blob/main/docs/docs/ns/Global/fc/assertEqual_LREAL.md *)
    VAR_INPUT
        act : LREAL; (*Variable to test*)
        xp : LREAL; (*Variable to test against*)
    END_VAR
END_FUNCTION
FUNCTION assertEqual_STRING : BOOL (* Returns TRUE if act = xp. *)(* https://github.com/tkucic/iecUnitTest/blob/main/docs/docs/ns/Global/fc/assertEqual_STRING.md *)
    VAR_INPUT
        act : STRING; (*Variable to test*)
        xp : STRING; (*Variable to test against*)
    END_VAR
END_FUNCTION
FUNCTION assertEqual_WSTRING : BOOL (* Returns TRUE if act = xp. *)(* https://github.com/tkucic/iecUnitTest/blob/main/docs/docs/ns/Global/fc/assertEqual_WSTRING.md *)
    VAR_INPUT
        act : wstring; (*Variable to test*)
        xp : wstring; (*Variable to test against*)
    END_VAR
END_FUNCTION
FUNCTION assertEqual_TIME : BOOL (* Returns TRUE if act = xp. *)(* https://github.com/tkucic/iecUnitTest/blob/main/docs/docs/ns/Global/fc/assertEqual_TIME.md *)
    VAR_INPUT
        act : TIME; (*Variable to test*)
        xp : TIME; (*Variable to test against*)
    END_VAR
END_FUNCTION
FUNCTION assertEqual_LTIME : BOOL (* Returns TRUE if act = xp. *)(* https://github.com/tkucic/iecUnitTest/blob/main/docs/docs/ns/Global/fc/assertEqual_LTIME.md *)
    VAR_INPUT
        act : LTIME; (*Variable to test*)
        xp : LTIME; (*Variable to test against*)
    END_VAR
END_FUNCTION
FUNCTION assertEqual_DATE : BOOL (* Returns TRUE if act = xp. *)(* https://github.com/tkucic/iecUnitTest/blob/main/docs/docs/ns/Global/fc/assertEqual_DATE.md *)
    VAR_INPUT
        act : DATE; (*Variable to test*)
        xp : DATE; (*Variable to test against*)
    END_VAR
END_FUNCTION
FUNCTION assertEqual_LDATE : BOOL (* Returns TRUE if act = xp. *)(* https://github.com/tkucic/iecUnitTest/blob/main/docs/docs/ns/Global/fc/assertEqual_LDATE.md *)
    VAR_INPUT
        act : LDATE; (*Variable to test*)
        xp : LDATE; (*Variable to test against*)
    END_VAR
END_FUNCTION
FUNCTION assertEqual_DATE_AND_TIME : BOOL (* Returns TRUE if act = xp. *)(* https://github.com/tkucic/iecUnitTest/blob/main/docs/docs/ns/Global/fc/assertEqual_DATE_AND_TIME.md *)
    VAR_INPUT
        act : DT; (*Variable to test*)
        xp : DT; (*Variable to test against*)
    END_VAR
END_FUNCTION
FUNCTION assertEqual_LDATE_AND_TIME : BOOL (* Returns TRUE if act = xp. *)(* https://github.com/tkucic/iecUnitTest/blob/main/docs/docs/ns/Global/fc/assertEqual_LDATE_AND_TIME.md *)
    VAR_INPUT
        act : LDATE_AND_TIME; (*Variable to test*)
        xp : LDATE_AND_TIME; (*Variable to test against*)
    END_VAR
END_FUNCTION
FUNCTION assertEqual_TIME_OF_DAY : BOOL (* Returns TRUE if act = xp. *)(* https://github.com/tkucic/iecUnitTest/blob/main/docs/docs/ns/Global/fc/assertEqual_TIME_OF_DAY.md *)
    VAR_INPUT
        act : TOD; (*Variable to test*)
        xp : TOD; (*Variable to test against*)
    END_VAR
END_FUNCTION
FUNCTION assertEqual_LTIME_OF_DAY : BOOL (* Returns TRUE if act = xp. *)(* https://github.com/tkucic/iecUnitTest/blob/main/docs/docs/ns/Global/fc/assertEqual_LTIME_OF_DAY.md *)
    VAR_INPUT
        act : LTIME_OF_DAY; (*Variable to test*)
        xp : LTIME_OF_DAY; (*Variable to test against*)
    END_VAR
END_FUNCTION
FUNCTION assertNotEqual_BOOL : BOOL (* Returns TRUE if act <> xp. *)(* https://github.com/tkucic/iecUnitTest/blob/main/docs/docs/ns/Global/fc/assertNotEqual_BOOL.md *)
    VAR_INPUT
        act : BOOL; (*Variable to test*)
        xp : BOOL; (*Variable to test against*)
    END_VAR
END_FUNCTION
FUNCTION assertNotEqual_BYTE : BOOL (* Returns TRUE if act <> xp. *)(* https://github.com/tkucic/iecUnitTest/blob/main/docs/docs/ns/Global/fc/assertNotEqual_BYTE.md *)
    VAR_INPUT
        act : BYTE; (*Variable to test*)
        xp : BYTE; (*Variable to test against*)
    END_VAR
END_FUNCTION
FUNCTION assertNotEqual_WORD : BOOL (* Returns TRUE if act <> xp. *)(* https://github.com/tkucic/iecUnitTest/blob/main/docs/docs/ns/Global/fc/assertNotEqual_WORD.md *)
    VAR_INPUT
        act : WORD; (*Variable to test*)
        xp : WORD; (*Variable to test against*)
    END_VAR
END_FUNCTION
FUNCTION assertNotEqual_DWORD : BOOL (* Returns TRUE if act <> xp. *)(* https://github.com/tkucic/iecUnitTest/blob/main/docs/docs/ns/Global/fc/assertNotEqual_DWORD.md *)
    VAR_INPUT
        act : DWORD; (*Variable to test*)
        xp : DWORD; (*Variable to test against*)
    END_VAR
END_FUNCTION
FUNCTION assertNotEqual_LWORD : BOOL (* Returns TRUE if act <> xp. *)(* https://github.com/tkucic/iecUnitTest/blob/main/docs/docs/ns/Global/fc/assertNotEqual_LWORD.md *)
    VAR_INPUT
        act : LWORD; (*Variable to test*)
        xp : LWORD; (*Variable to test against*)
    END_VAR
END_FUNCTION
FUNCTION assertNotEqual_SINT : BOOL (* Returns TRUE if act <> xp. *)(* https://github.com/tkucic/iecUnitTest/blob/main/docs/docs/ns/Global/fc/assertNotEqual_SINT.md *)
    VAR_INPUT
        act : SINT; (*Variable to test*)
        xp : SINT; (*Variable to test against*)
    END_VAR
END_FUNCTION
FUNCTION assertNotEqual_USINT : BOOL (* Returns TRUE if act <> xp. *)(* https://github.com/tkucic/iecUnitTest/blob/main/docs/docs/ns/Global/fc/assertNotEqual_USINT.md *)
    VAR_INPUT
        act : USINT; (*Variable to test*)
        xp : USINT; (*Variable to test against*)
    END_VAR
END_FUNCTION
FUNCTION assertNotEqual_INT : BOOL (* Returns TRUE if act <> xp. *)(* https://github.com/tkucic/iecUnitTest/blob/main/docs/docs/ns/Global/fc/assertNotEqual_INT.md *)
    VAR_INPUT
        act : INT; (*Variable to test*)
        xp : INT; (*Variable to test against*)
    END_VAR
END_FUNCTION
FUNCTION assertNotEqual_UINT : BOOL (* Returns TRUE if act <> xp. *)(* https://github.com/tkucic/iecUnitTest/blob/main/docs/docs/ns/Global/fc/assertNotEqual_UINT.md *)
    VAR_INPUT
        act : UINT; (*Variable to test*)
        xp : UINT; (*Variable to test against*)
    END_VAR
END_FUNCTION
FUNCTION assertNotEqual_DINT : BOOL (* Returns TRUE if act <> xp. *)(* https://github.com/tkucic/iecUnitTest/blob/main/docs/docs/ns/Global/fc/assertNotEqual_DINT.md *)
    VAR_INPUT
        act : DINT; (*Variable to test*)
        xp : DINT; (*Variable to test against*)
    END_VAR
END_FUNCTION
FUNCTION assertNotEqual_UDINT : BOOL (* Returns TRUE if act <> xp. *)(* https://github.com/tkucic/iecUnitTest/blob/main/docs/docs/ns/Global/fc/assertNotEqual_UDINT.md *)
    VAR_INPUT
        act : UDINT; (*Variable to test*)
        xp : UDINT; (*Variable to test against*)
    END_VAR
END_FUNCTION
FUNCTION assertNotEqual_LINT : BOOL (* Returns TRUE if act <> xp. *)(* https://github.com/tkucic/iecUnitTest/blob/main/docs/docs/ns/Global/fc/assertNotEqual_LINT.md *)
    VAR_INPUT
        act : LINT; (*Variable to test*)
        xp : LINT; (*Variable to test against*)
    END_VAR
END_FUNCTION
FUNCTION assertNotEqual_ULINT : BOOL (* Returns TRUE if act <> xp. *)(* https://github.com/tkucic/iecUnitTest/blob/main/docs/docs/ns/Global/fc/assertNotEqual_ULINT.md *)
    VAR_INPUT
        act : ULINT; (*Variable to test*)
        xp : ULINT; (*Variable to test against*)
    END_VAR
END_FUNCTION
FUNCTION assertNotEqual_REAL : BOOL (* Returns TRUE if act <> xp. *)(* https://github.com/tkucic/iecUnitTest/blob/main/docs/docs/ns/Global/fc/assertNotEqual_REAL.md *)
    VAR_INPUT
        act : REAL; (*Variable to test*)
        xp : REAL; (*Variable to test against*)
    END_VAR
END_FUNCTION
FUNCTION assertNotEqual_LREAL : BOOL (* Returns TRUE if act <> xp. *)(* https://github.com/tkucic/iecUnitTest/blob/main/docs/docs/ns/Global/fc/assertNotEqual_LREAL.md *)
    VAR_INPUT
        act : LREAL; (*Variable to test*)
        xp : LREAL; (*Variable to test against*)
    END_VAR
END_FUNCTION
FUNCTION assertNotEqual_STRING : BOOL (* Returns TRUE if act <> xp. *)(* https://github.com/tkucic/iecUnitTest/blob/main/docs/docs/ns/Global/fc/assertNotEqual_STRING.md *)
    VAR_INPUT
        act : STRING; (*Variable to test*)
        xp : STRING; (*Variable to test against*)
    END_VAR
END_FUNCTION
FUNCTION assertNotEqual_WSTRING : BOOL (* Returns TRUE if act <> xp. *)(* https://github.com/tkucic/iecUnitTest/blob/main/docs/docs/ns/Global/fc/assertNotEqual_WSTRING.md *)
    VAR_INPUT
        act : wstring; (*Variable to test*)
        xp : wstring; (*Variable to test against*)
    END_VAR
END_FUNCTION
FUNCTION assertNotEqual_TIME : BOOL (* Returns TRUE if act <> xp. *)(* https://github.com/tkucic/iecUnitTest/blob/main/docs/docs/ns/Global/fc/assertNotEqual_TIME.md *)
    VAR_INPUT
        act : TIME; (*Variable to test*)
        xp : TIME; (*Variable to test against*)
    END_VAR
END_FUNCTION
FUNCTION assertNotEqual_LTIME : BOOL (* Returns TRUE if act <> xp. *)(* https://github.com/tkucic/iecUnitTest/blob/main/docs/docs/ns/Global/fc/assertNotEqual_LTIME.md *)
    VAR_INPUT
        act : LTIME; (*Variable to test*)
        xp : LTIME; (*Variable to test against*)
    END_VAR
END_FUNCTION
FUNCTION assertNotEqual_DATE : BOOL (* Returns TRUE if act <> xp. *)(* https://github.com/tkucic/iecUnitTest/blob/main/docs/docs/ns/Global/fc/assertNotEqual_DATE.md *)
    VAR_INPUT
        act : DATE; (*Variable to test*)
        xp : DATE; (*Variable to test against*)
    END_VAR
END_FUNCTION
FUNCTION assertNotEqual_LDATE : BOOL (* Returns TRUE if act <> xp. *)(* https://github.com/tkucic/iecUnitTest/blob/main/docs/docs/ns/Global/fc/assertNotEqual_LDATE.md *)
    VAR_INPUT
        act : LDATE; (*Variable to test*)
        xp : LDATE; (*Variable to test against*)
    END_VAR
END_FUNCTION
FUNCTION assertNotEqual_DATE_AND_TIME : BOOL (* Returns TRUE if act <> xp. *)(* https://github.com/tkucic/iecUnitTest/blob/main/docs/docs/ns/Global/fc/assertNotEqual_DATE_AND_TIME.md *)
    VAR_INPUT
        act : DT; (*Variable to test*)
        xp : DT; (*Variable to test against*)
    END_VAR
END_FUNCTION
FUNCTION assertNotEqual_LDATE_AND_TIME : BOOL (* Returns TRUE if act <> xp. *)(* https://github.com/tkucic/iecUnitTest/blob/main/docs/docs/ns/Global/fc/assertNotEqual_LDATE_AND_TIME.md *)
    VAR_INPUT
        act : LDATE_AND_TIME; (*Variable to test*)
        xp : LDATE_AND_TIME; (*Variable to test against*)
    END_VAR
END_FUNCTION
FUNCTION assertNotEqual_TIME_OF_DAY : BOOL (* Returns TRUE if act <> xp. *)(* https://github.com/tkucic/iecUnitTest/blob/main/docs/docs/ns/Global/fc/assertNotEqual_TIME_OF_DAY.md *)
    VAR_INPUT
        act : TOD; (*Variable to test*)
        xp : TOD; (*Variable to test against*)
    END_VAR
END_FUNCTION
FUNCTION assertNotEqual_LTIME_OF_DAY : BOOL (* Returns TRUE if act <> xp. *)(* https://github.com/tkucic/iecUnitTest/blob/main/docs/docs/ns/Global/fc/assertNotEqual_LTIME_OF_DAY.md *)
    VAR_INPUT
        act : LTIME_OF_DAY; (*Variable to test*)
        xp : LTIME_OF_DAY; (*Variable to test against*)
    END_VAR
END_FUNCTION
FUNCTION assertGreater_BYTE : BOOL (* Returns TRUE if act > xp. *)(* https://github.com/tkucic/iecUnitTest/blob/main/docs/docs/ns/Global/fc/assertGreater_BYTE.md *)
    VAR_INPUT
        act : BYTE; (*Variable to test*)
        xp : BYTE; (*Variable to test against*)
    END_VAR
END_FUNCTION
FUNCTION assertGreater_WORD : BOOL (* Returns TRUE if act > xp. *)(* https://github.com/tkucic/iecUnitTest/blob/main/docs/docs/ns/Global/fc/assertGreater_WORD.md *)
    VAR_INPUT
        act : WORD; (*Variable to test*)
        xp : WORD; (*Variable to test against*)
    END_VAR
END_FUNCTION
FUNCTION assertGreater_DWORD : BOOL (* Returns TRUE if act > xp. *)(* https://github.com/tkucic/iecUnitTest/blob/main/docs/docs/ns/Global/fc/assertGreater_DWORD.md *)
    VAR_INPUT
        act : DWORD; (*Variable to test*)
        xp : DWORD; (*Variable to test against*)
    END_VAR
END_FUNCTION
FUNCTION assertGreater_LWORD : BOOL (* Returns TRUE if act > xp. *)(* https://github.com/tkucic/iecUnitTest/blob/main/docs/docs/ns/Global/fc/assertGreater_LWORD.md *)
    VAR_INPUT
        act : LWORD; (*Variable to test*)
        xp : LWORD; (*Variable to test against*)
    END_VAR
END_FUNCTION
FUNCTION assertGreater_SINT : BOOL (* Returns TRUE if act > xp. *)(* https://github.com/tkucic/iecUnitTest/blob/main/docs/docs/ns/Global/fc/assertGreater_SINT.md *)
    VAR_INPUT
        act : SINT; (*Variable to test*)
        xp : SINT; (*Variable to test against*)
    END_VAR
END_FUNCTION
FUNCTION assertGreater_USINT : BOOL (* Returns TRUE if act > xp. *)(* https://github.com/tkucic/iecUnitTest/blob/main/docs/docs/ns/Global/fc/assertGreater_USINT.md *)
    VAR_INPUT
        act : USINT; (*Variable to test*)
        xp : USINT; (*Variable to test against*)
    END_VAR
END_FUNCTION
FUNCTION assertGreater_INT : BOOL (* Returns TRUE if act > xp. *)(* https://github.com/tkucic/iecUnitTest/blob/main/docs/docs/ns/Global/fc/assertGreater_INT.md *)
    VAR_INPUT
        act : INT; (*Variable to test*)
        xp : INT; (*Variable to test against*)
    END_VAR
END_FUNCTION
FUNCTION assertGreater_UINT : BOOL (* Returns TRUE if act > xp. *)(* https://github.com/tkucic/iecUnitTest/blob/main/docs/docs/ns/Global/fc/assertGreater_UINT.md *)
    VAR_INPUT
        act : UINT; (*Variable to test*)
        xp : UINT; (*Variable to test against*)
    END_VAR
END_FUNCTION
FUNCTION assertGreater_DINT : BOOL (* Returns TRUE if act > xp. *)(* https://github.com/tkucic/iecUnitTest/blob/main/docs/docs/ns/Global/fc/assertGreater_DINT.md *)
    VAR_INPUT
        act : DINT; (*Variable to test*)
        xp : DINT; (*Variable to test against*)
    END_VAR
END_FUNCTION
FUNCTION assertGreater_UDINT : BOOL (* Returns TRUE if act > xp. *)(* https://github.com/tkucic/iecUnitTest/blob/main/docs/docs/ns/Global/fc/assertGreater_UDINT.md *)
    VAR_INPUT
        act : UDINT; (*Variable to test*)
        xp : UDINT; (*Variable to test against*)
    END_VAR
END_FUNCTION
FUNCTION assertGreater_LINT : BOOL (* Returns TRUE if act > xp. *)(* https://github.com/tkucic/iecUnitTest/blob/main/docs/docs/ns/Global/fc/assertGreater_LINT.md *)
    VAR_INPUT
        act : LINT; (*Variable to test*)
        xp : LINT; (*Variable to test against*)
    END_VAR
END_FUNCTION
FUNCTION assertGreater_ULINT : BOOL (* Returns TRUE if act > xp. *)(* https://github.com/tkucic/iecUnitTest/blob/main/docs/docs/ns/Global/fc/assertGreater_ULINT.md *)
    VAR_INPUT
        act : ULINT; (*Variable to test*)
        xp : ULINT; (*Variable to test against*)
    END_VAR
END_FUNCTION
FUNCTION assertGreater_REAL : BOOL (* Returns TRUE if act > xp. *)(* https://github.com/tkucic/iecUnitTest/blob/main/docs/docs/ns/Global/fc/assertGreater_REAL.md *)
    VAR_INPUT
        act : REAL; (*Variable to test*)
        xp : REAL; (*Variable to test against*)
    END_VAR
END_FUNCTION
FUNCTION assertGreater_LREAL : BOOL (* Returns TRUE if act > xp. *)(* https://github.com/tkucic/iecUnitTest/blob/main/docs/docs/ns/Global/fc/assertGreater_LREAL.md *)
    VAR_INPUT
        act : LREAL; (*Variable to test*)
        xp : LREAL; (*Variable to test against*)
    END_VAR
END_FUNCTION
FUNCTION assertGreater_TIME : BOOL (* Returns TRUE if act > xp. *)(* https://github.com/tkucic/iecUnitTest/blob/main/docs/docs/ns/Global/fc/assertGreater_TIME.md *)
    VAR_INPUT
        act : TIME; (*Variable to test*)
        xp : TIME; (*Variable to test against*)
    END_VAR
END_FUNCTION
FUNCTION assertGreater_LTIME : BOOL (* Returns TRUE if act > xp. *)(* https://github.com/tkucic/iecUnitTest/blob/main/docs/docs/ns/Global/fc/assertGreater_LTIME.md *)
    VAR_INPUT
        act : LTIME; (*Variable to test*)
        xp : LTIME; (*Variable to test against*)
    END_VAR
END_FUNCTION
FUNCTION assertGreater_DATE : BOOL (* Returns TRUE if act > xp. *)(* https://github.com/tkucic/iecUnitTest/blob/main/docs/docs/ns/Global/fc/assertGreater_DATE.md *)
    VAR_INPUT
        act : DATE; (*Variable to test*)
        xp : DATE; (*Variable to test against*)
    END_VAR
END_FUNCTION
FUNCTION assertGreater_LDATE : BOOL (* Returns TRUE if act > xp. *)(* https://github.com/tkucic/iecUnitTest/blob/main/docs/docs/ns/Global/fc/assertGreater_LDATE.md *)
    VAR_INPUT
        act : LDATE; (*Variable to test*)
        xp : LDATE; (*Variable to test against*)
    END_VAR
END_FUNCTION
FUNCTION assertGreater_DATE_AND_TIME : BOOL (* Returns TRUE if act > xp. *)(* https://github.com/tkucic/iecUnitTest/blob/main/docs/docs/ns/Global/fc/assertGreater_DATE_AND_TIME.md *)
    VAR_INPUT
        act : DT; (*Variable to test*)
        xp : DT; (*Variable to test against*)
    END_VAR
END_FUNCTION
FUNCTION assertGreater_LDATE_AND_TIME : BOOL (* Returns TRUE if act > xp. *)(* https://github.com/tkucic/iecUnitTest/blob/main/docs/docs/ns/Global/fc/assertGreater_LDATE_AND_TIME.md *)
    VAR_INPUT
        act : LDATE_AND_TIME; (*Variable to test*)
        xp : LDATE_AND_TIME; (*Variable to test against*)
    END_VAR
END_FUNCTION
FUNCTION assertGreater_TIME_OF_DAY : BOOL (* Returns TRUE if act > xp. *)(* https://github.com/tkucic/iecUnitTest/blob/main/docs/docs/ns/Global/fc/assertGreater_TIME_OF_DAY.md *)
    VAR_INPUT
        act : TOD; (*Variable to test*)
        xp : TOD; (*Variable to test against*)
    END_VAR
END_FUNCTION
FUNCTION assertGreater_LTIME_OF_DAY : BOOL (* Returns TRUE if act > xp. *)(* https://github.com/tkucic/iecUnitTest/blob/main/docs/docs/ns/Global/fc/assertGreater_LTIME_OF_DAY.md *)
    VAR_INPUT
        act : LTIME_OF_DAY; (*Variable to test*)
        xp : LTIME_OF_DAY; (*Variable to test against*)
    END_VAR
END_FUNCTION
FUNCTION assertGreaterEqual_BYTE : BOOL (* Returns TRUE if act >= xp. *)(* https://github.com/tkucic/iecUnitTest/blob/main/docs/docs/ns/Global/fc/assertGreaterEqual_BYTE.md *)
    VAR_INPUT
        act : BYTE; (*Variable to test*)
        xp : BYTE; (*Variable to test against*)
    END_VAR
END_FUNCTION
FUNCTION assertGreaterEqual_WORD : BOOL (* Returns TRUE if act >= xp. *)(* https://github.com/tkucic/iecUnitTest/blob/main/docs/docs/ns/Global/fc/assertGreaterEqual_WORD.md *)
    VAR_INPUT
        act : WORD; (*Variable to test*)
        xp : WORD; (*Variable to test against*)
    END_VAR
END_FUNCTION
FUNCTION assertGreaterEqual_DWORD : BOOL (* Returns TRUE if act >= xp. *)(* https://github.com/tkucic/iecUnitTest/blob/main/docs/docs/ns/Global/fc/assertGreaterEqual_DWORD.md *)
    VAR_INPUT
        act : DWORD; (*Variable to test*)
        xp : DWORD; (*Variable to test against*)
    END_VAR
END_FUNCTION
FUNCTION assertGreaterEqual_LWORD : BOOL (* Returns TRUE if act >= xp. *)(* https://github.com/tkucic/iecUnitTest/blob/main/docs/docs/ns/Global/fc/assertGreaterEqual_LWORD.md *)
    VAR_INPUT
        act : LWORD; (*Variable to test*)
        xp : LWORD; (*Variable to test against*)
    END_VAR
END_FUNCTION
FUNCTION assertGreaterEqual_SINT : BOOL (* Returns TRUE if act >= xp. *)(* https://github.com/tkucic/iecUnitTest/blob/main/docs/docs/ns/Global/fc/assertGreaterEqual_SINT.md *)
    VAR_INPUT
        act : SINT; (*Variable to test*)
        xp : SINT; (*Variable to test against*)
    END_VAR
END_FUNCTION
FUNCTION assertGreaterEqual_USINT : BOOL (* Returns TRUE if act >= xp. *)(* https://github.com/tkucic/iecUnitTest/blob/main/docs/docs/ns/Global/fc/assertGreaterEqual_USINT.md *)
    VAR_INPUT
        act : USINT; (*Variable to test*)
        xp : USINT; (*Variable to test against*)
    END_VAR
END_FUNCTION
FUNCTION assertGreaterEqual_INT : BOOL (* Returns TRUE if act >= xp. *)(* https://github.com/tkucic/iecUnitTest/blob/main/docs/docs/ns/Global/fc/assertGreaterEqual_INT.md *)
    VAR_INPUT
        act : INT; (*Variable to test*)
        xp : INT; (*Variable to test against*)
    END_VAR
END_FUNCTION
FUNCTION assertGreaterEqual_UINT : BOOL (* Returns TRUE if act >= xp. *)(* https://github.com/tkucic/iecUnitTest/blob/main/docs/docs/ns/Global/fc/assertGreaterEqual_UINT.md *)
    VAR_INPUT
        act : UINT; (*Variable to test*)
        xp : UINT; (*Variable to test against*)
    END_VAR
END_FUNCTION
FUNCTION assertGreaterEqual_DINT : BOOL (* Returns TRUE if act >= xp. *)(* https://github.com/tkucic/iecUnitTest/blob/main/docs/docs/ns/Global/fc/assertGreaterEqual_DINT.md *)
    VAR_INPUT
        act : DINT; (*Variable to test*)
        xp : DINT; (*Variable to test against*)
    END_VAR
END_FUNCTION
FUNCTION assertGreaterEqual_UDINT : BOOL (* Returns TRUE if act >= xp. *)(* https://github.com/tkucic/iecUnitTest/blob/main/docs/docs/ns/Global/fc/assertGreaterEqual_UDINT.md *)
    VAR_INPUT
        act : UDINT; (*Variable to test*)
        xp : UDINT; (*Variable to test against*)
    END_VAR
END_FUNCTION
FUNCTION assertGreaterEqual_LINT : BOOL (* Returns TRUE if act >= xp. *)(* https://github.com/tkucic/iecUnitTest/blob/main/docs/docs/ns/Global/fc/assertGreaterEqual_LINT.md *)
    VAR_INPUT
        act : LINT; (*Variable to test*)
        xp : LINT; (*Variable to test against*)
    END_VAR
END_FUNCTION
FUNCTION assertGreaterEqual_ULINT : BOOL (* Returns TRUE if act >= xp. *)(* https://github.com/tkucic/iecUnitTest/blob/main/docs/docs/ns/Global/fc/assertGreaterEqual_ULINT.md *)
    VAR_INPUT
        act : ULINT; (*Variable to test*)
        xp : ULINT; (*Variable to test against*)
    END_VAR
END_FUNCTION
FUNCTION assertGreaterEqual_REAL : BOOL (* Returns TRUE if act >= xp. *)(* https://github.com/tkucic/iecUnitTest/blob/main/docs/docs/ns/Global/fc/assertGreaterEqual_REAL.md *)
    VAR_INPUT
        act : REAL; (*Variable to test*)
        xp : REAL; (*Variable to test against*)
    END_VAR
END_FUNCTION
FUNCTION assertGreaterEqual_LREAL : BOOL (* Returns TRUE if act >= xp. *)(* https://github.com/tkucic/iecUnitTest/blob/main/docs/docs/ns/Global/fc/assertGreaterEqual_LREAL.md *)
    VAR_INPUT
        act : LREAL; (*Variable to test*)
        xp : LREAL; (*Variable to test against*)
    END_VAR
END_FUNCTION
FUNCTION assertGreaterEqual_TIME : BOOL (* Returns TRUE if act >= xp. *)(* https://github.com/tkucic/iecUnitTest/blob/main/docs/docs/ns/Global/fc/assertGreaterEqual_TIME.md *)
    VAR_INPUT
        act : TIME; (*Variable to test*)
        xp : TIME; (*Variable to test against*)
    END_VAR
END_FUNCTION
FUNCTION assertGreaterEqual_LTIME : BOOL (* Returns TRUE if act >= xp. *)(* https://github.com/tkucic/iecUnitTest/blob/main/docs/docs/ns/Global/fc/assertGreaterEqual_LTIME.md *)
    VAR_INPUT
        act : LTIME; (*Variable to test*)
        xp : LTIME; (*Variable to test against*)
    END_VAR
END_FUNCTION
FUNCTION assertGreaterEqual_DATE : BOOL (* Returns TRUE if act >= xp. *)(* https://github.com/tkucic/iecUnitTest/blob/main/docs/docs/ns/Global/fc/assertGreaterEqual_DATE.md *)
    VAR_INPUT
        act : DATE; (*Variable to test*)
        xp : DATE; (*Variable to test against*)
    END_VAR
END_FUNCTION
FUNCTION assertGreaterEqual_LDATE : BOOL (* Returns TRUE if act >= xp. *)(* https://github.com/tkucic/iecUnitTest/blob/main/docs/docs/ns/Global/fc/assertGreaterEqual_LDATE.md *)
    VAR_INPUT
        act : LDATE; (*Variable to test*)
        xp : LDATE; (*Variable to test against*)
    END_VAR
END_FUNCTION
FUNCTION assertGreaterEqual_DATE_AND_TIME : BOOL (* Returns TRUE if act >= xp. *)(* https://github.com/tkucic/iecUnitTest/blob/main/docs/docs/ns/Global/fc/assertGreaterEqual_DATE_AND_TIME.md *)
    VAR_INPUT
        act : DT; (*Variable to test*)
        xp : DT; (*Variable to test against*)
    END_VAR
END_FUNCTION
FUNCTION assertGreaterEqual_LDATE_AND_TIME : BOOL (* Returns TRUE if act >= xp. *)(* https://github.com/tkucic/iecUnitTest/blob/main/docs/docs/ns/Global/fc/assertGreaterEqual_LDATE_AND_TIME.md *)
    VAR_INPUT
        act : LDATE_AND_TIME; (*Variable to test*)
        xp : LDATE_AND_TIME; (*Variable to test against*)
    END_VAR
END_FUNCTION
FUNCTION assertGreaterEqual_TIME_OF_DAY : BOOL (* Returns TRUE if act >= xp. *)(* https://github.com/tkucic/iecUnitTest/blob/main/docs/docs/ns/Global/fc/assertGreaterEqual_TIME_OF_DAY.md *)
    VAR_INPUT
        act : TOD; (*Variable to test*)
        xp : TOD; (*Variable to test against*)
    END_VAR
END_FUNCTION
FUNCTION assertGreaterEqual_LTIME_OF_DAY : BOOL (* Returns TRUE if act >= xp. *)(* https://github.com/tkucic/iecUnitTest/blob/main/docs/docs/ns/Global/fc/assertGreaterEqual_LTIME_OF_DAY.md *)
    VAR_INPUT
        act : LTIME_OF_DAY; (*Variable to test*)
        xp : LTIME_OF_DAY; (*Variable to test against*)
    END_VAR
END_FUNCTION
FUNCTION assertLess_BYTE : BOOL (* Returns TRUE if act < xp. *)(* https://github.com/tkucic/iecUnitTest/blob/main/docs/docs/ns/Global/fc/assertLess_BYTE.md *)
    VAR_INPUT
        act : BYTE; (*Variable to test*)
        xp : BYTE; (*Variable to test against*)
    END_VAR
END_FUNCTION
FUNCTION assertLess_WORD : BOOL (* Returns TRUE if act < xp. *)(* https://github.com/tkucic/iecUnitTest/blob/main/docs/docs/ns/Global/fc/assertLess_WORD.md *)
    VAR_INPUT
        act : WORD; (*Variable to test*)
        xp : WORD; (*Variable to test against*)
    END_VAR
END_FUNCTION
FUNCTION assertLess_DWORD : BOOL (* Returns TRUE if act < xp. *)(* https://github.com/tkucic/iecUnitTest/blob/main/docs/docs/ns/Global/fc/assertLess_DWORD.md *)
    VAR_INPUT
        act : DWORD; (*Variable to test*)
        xp : DWORD; (*Variable to test against*)
    END_VAR
END_FUNCTION
FUNCTION assertLess_LWORD : BOOL (* Returns TRUE if act < xp. *)(* https://github.com/tkucic/iecUnitTest/blob/main/docs/docs/ns/Global/fc/assertLess_LWORD.md *)
    VAR_INPUT
        act : LWORD; (*Variable to test*)
        xp : LWORD; (*Variable to test against*)
    END_VAR
END_FUNCTION
FUNCTION assertLess_SINT : BOOL (* Returns TRUE if act < xp. *)(* https://github.com/tkucic/iecUnitTest/blob/main/docs/docs/ns/Global/fc/assertLess_SINT.md *)
    VAR_INPUT
        act : SINT; (*Variable to test*)
        xp : SINT; (*Variable to test against*)
    END_VAR
END_FUNCTION
FUNCTION assertLess_USINT : BOOL (* Returns TRUE if act < xp. *)(* https://github.com/tkucic/iecUnitTest/blob/main/docs/docs/ns/Global/fc/assertLess_USINT.md *)
    VAR_INPUT
        act : USINT; (*Variable to test*)
        xp : USINT; (*Variable to test against*)
    END_VAR
END_FUNCTION
FUNCTION assertLess_INT : BOOL (* Returns TRUE if act < xp. *)(* https://github.com/tkucic/iecUnitTest/blob/main/docs/docs/ns/Global/fc/assertLess_INT.md *)
    VAR_INPUT
        act : INT; (*Variable to test*)
        xp : INT; (*Variable to test against*)
    END_VAR
END_FUNCTION
FUNCTION assertLess_UINT : BOOL (* Returns TRUE if act < xp. *)(* https://github.com/tkucic/iecUnitTest/blob/main/docs/docs/ns/Global/fc/assertLess_UINT.md *)
    VAR_INPUT
        act : UINT; (*Variable to test*)
        xp : UINT; (*Variable to test against*)
    END_VAR
END_FUNCTION
FUNCTION assertLess_DINT : BOOL (* Returns TRUE if act < xp. *)(* https://github.com/tkucic/iecUnitTest/blob/main/docs/docs/ns/Global/fc/assertLess_DINT.md *)
    VAR_INPUT
        act : DINT; (*Variable to test*)
        xp : DINT; (*Variable to test against*)
    END_VAR
END_FUNCTION
FUNCTION assertLess_UDINT : BOOL (* Returns TRUE if act < xp. *)(* https://github.com/tkucic/iecUnitTest/blob/main/docs/docs/ns/Global/fc/assertLess_UDINT.md *)
    VAR_INPUT
        act : UDINT; (*Variable to test*)
        xp : UDINT; (*Variable to test against*)
    END_VAR
END_FUNCTION
FUNCTION assertLess_LINT : BOOL (* Returns TRUE if act < xp. *)(* https://github.com/tkucic/iecUnitTest/blob/main/docs/docs/ns/Global/fc/assertLess_LINT.md *)
    VAR_INPUT
        act : LINT; (*Variable to test*)
        xp : LINT; (*Variable to test against*)
    END_VAR
END_FUNCTION
FUNCTION assertLess_ULINT : BOOL (* Returns TRUE if act < xp. *)(* https://github.com/tkucic/iecUnitTest/blob/main/docs/docs/ns/Global/fc/assertLess_ULINT.md *)
    VAR_INPUT
        act : ULINT; (*Variable to test*)
        xp : ULINT; (*Variable to test against*)
    END_VAR
END_FUNCTION
FUNCTION assertLess_REAL : BOOL (* Returns TRUE if act < xp. *)(* https://github.com/tkucic/iecUnitTest/blob/main/docs/docs/ns/Global/fc/assertLess_REAL.md *)
    VAR_INPUT
        act : REAL; (*Variable to test*)
        xp : REAL; (*Variable to test against*)
    END_VAR
END_FUNCTION
FUNCTION assertLess_LREAL : BOOL (* Returns TRUE if act < xp. *)(* https://github.com/tkucic/iecUnitTest/blob/main/docs/docs/ns/Global/fc/assertLess_LREAL.md *)
    VAR_INPUT
        act : LREAL; (*Variable to test*)
        xp : LREAL; (*Variable to test against*)
    END_VAR
END_FUNCTION
FUNCTION assertLess_TIME : BOOL (* Returns TRUE if act < xp. *)(* https://github.com/tkucic/iecUnitTest/blob/main/docs/docs/ns/Global/fc/assertLess_TIME.md *)
    VAR_INPUT
        act : TIME; (*Variable to test*)
        xp : TIME; (*Variable to test against*)
    END_VAR
END_FUNCTION
FUNCTION assertLess_LTIME : BOOL (* Returns TRUE if act < xp. *)(* https://github.com/tkucic/iecUnitTest/blob/main/docs/docs/ns/Global/fc/assertLess_LTIME.md *)
    VAR_INPUT
        act : LTIME; (*Variable to test*)
        xp : LTIME; (*Variable to test against*)
    END_VAR
END_FUNCTION
FUNCTION assertLess_DATE : BOOL (* Returns TRUE if act < xp. *)(* https://github.com/tkucic/iecUnitTest/blob/main/docs/docs/ns/Global/fc/assertLess_DATE.md *)
    VAR_INPUT
        act : DATE; (*Variable to test*)
        xp : DATE; (*Variable to test against*)
    END_VAR
END_FUNCTION
FUNCTION assertLess_LDATE : BOOL (* Returns TRUE if act < xp. *)(* https://github.com/tkucic/iecUnitTest/blob/main/docs/docs/ns/Global/fc/assertLess_LDATE.md *)
    VAR_INPUT
        act : LDATE; (*Variable to test*)
        xp : LDATE; (*Variable to test against*)
    END_VAR
END_FUNCTION
FUNCTION assertLess_DATE_AND_TIME : BOOL (* Returns TRUE if act < xp. *)(* https://github.com/tkucic/iecUnitTest/blob/main/docs/docs/ns/Global/fc/assertLess_DATE_AND_TIME.md *)
    VAR_INPUT
        act : DT; (*Variable to test*)
        xp : DT; (*Variable to test against*)
    END_VAR
END_FUNCTION
FUNCTION assertLess_LDATE_AND_TIME : BOOL (* Returns TRUE if act < xp. *)(* https://github.com/tkucic/iecUnitTest/blob/main/docs/docs/ns/Global/fc/assertLess_LDATE_AND_TIME.md *)
    VAR_INPUT
        act : LDATE_AND_TIME; (*Variable to test*)
        xp : LDATE_AND_TIME; (*Variable to test against*)
    END_VAR
END_FUNCTION
FUNCTION assertLess_TIME_OF_DAY : BOOL (* Returns TRUE if act < xp. *)(* https://github.com/tkucic/iecUnitTest/blob/main/docs/docs/ns/Global/fc/assertLess_TIME_OF_DAY.md *)
    VAR_INPUT
        act : TOD; (*Variable to test*)
        xp : TOD; (*Variable to test against*)
    END_VAR
END_FUNCTION
FUNCTION assertLess_LTIME_OF_DAY : BOOL (* Returns TRUE if act < xp. *)(* https://github.com/tkucic/iecUnitTest/blob/main/docs/docs/ns/Global/fc/assertLess_LTIME_OF_DAY.md *)
    VAR_INPUT
        act : LTIME_OF_DAY; (*Variable to test*)
        xp : LTIME_OF_DAY; (*Variable to test against*)
    END_VAR
END_FUNCTION
FUNCTION assertLessEqual_BYTE : BOOL (* Returns TRUE if act <= xp. *)(* https://github.com/tkucic/iecUnitTest/blob/main/docs/docs/ns/Global/fc/assertLessEqual_BYTE.md *)
    VAR_INPUT
        act : BYTE; (*Variable to test*)
        xp : BYTE; (*Variable to test against*)
    END_VAR
END_FUNCTION
FUNCTION assertLessEqual_WORD : BOOL (* Returns TRUE if act <= xp. *)(* https://github.com/tkucic/iecUnitTest/blob/main/docs/docs/ns/Global/fc/assertLessEqual_WORD.md *)
    VAR_INPUT
        act : WORD; (*Variable to test*)
        xp : WORD; (*Variable to test against*)
    END_VAR
END_FUNCTION
FUNCTION assertLessEqual_DWORD : BOOL (* Returns TRUE if act <= xp. *)(* https://github.com/tkucic/iecUnitTest/blob/main/docs/docs/ns/Global/fc/assertLessEqual_DWORD.md *)
    VAR_INPUT
        act : DWORD; (*Variable to test*)
        xp : DWORD; (*Variable to test against*)
    END_VAR
END_FUNCTION
FUNCTION assertLessEqual_LWORD : BOOL (* Returns TRUE if act <= xp. *)(* https://github.com/tkucic/iecUnitTest/blob/main/docs/docs/ns/Global/fc/assertLessEqual_LWORD.md *)
    VAR_INPUT
        act : LWORD; (*Variable to test*)
        xp : LWORD; (*Variable to test against*)
    END_VAR
END_FUNCTION
FUNCTION assertLessEqual_SINT : BOOL (* Returns TRUE if act <= xp. *)(* https://github.com/tkucic/iecUnitTest/blob/main/docs/docs/ns/Global/fc/assertLessEqual_SINT.md *)
    VAR_INPUT
        act : SINT; (*Variable to test*)
        xp : SINT; (*Variable to test against*)
    END_VAR
END_FUNCTION
FUNCTION assertLessEqual_USINT : BOOL (* Returns TRUE if act <= xp. *)(* https://github.com/tkucic/iecUnitTest/blob/main/docs/docs/ns/Global/fc/assertLessEqual_USINT.md *)
    VAR_INPUT
        act : USINT; (*Variable to test*)
        xp : USINT; (*Variable to test against*)
    END_VAR
END_FUNCTION
FUNCTION assertLessEqual_INT : BOOL (* Returns TRUE if act <= xp. *)(* https://github.com/tkucic/iecUnitTest/blob/main/docs/docs/ns/Global/fc/assertLessEqual_INT.md *)
    VAR_INPUT
        act : INT; (*Variable to test*)
        xp : INT; (*Variable to test against*)
    END_VAR
END_FUNCTION
FUNCTION assertLessEqual_UINT : BOOL (* Returns TRUE if act <= xp. *)(* https://github.com/tkucic/iecUnitTest/blob/main/docs/docs/ns/Global/fc/assertLessEqual_UINT.md *)
    VAR_INPUT
        act : UINT; (*Variable to test*)
        xp : UINT; (*Variable to test against*)
    END_VAR
END_FUNCTION
FUNCTION assertLessEqual_DINT : BOOL (* Returns TRUE if act <= xp. *)(* https://github.com/tkucic/iecUnitTest/blob/main/docs/docs/ns/Global/fc/assertLessEqual_DINT.md *)
    VAR_INPUT
        act : DINT; (*Variable to test*)
        xp : DINT; (*Variable to test against*)
    END_VAR
END_FUNCTION
FUNCTION assertLessEqual_UDINT : BOOL (* Returns TRUE if act <= xp. *)(* https://github.com/tkucic/iecUnitTest/blob/main/docs/docs/ns/Global/fc/assertLessEqual_UDINT.md *)
    VAR_INPUT
        act : UDINT; (*Variable to test*)
        xp : UDINT; (*Variable to test against*)
    END_VAR
END_FUNCTION
FUNCTION assertLessEqual_LINT : BOOL (* Returns TRUE if act <= xp. *)(* https://github.com/tkucic/iecUnitTest/blob/main/docs/docs/ns/Global/fc/assertLessEqual_LINT.md *)
    VAR_INPUT
        act : LINT; (*Variable to test*)
        xp : LINT; (*Variable to test against*)
    END_VAR
END_FUNCTION
FUNCTION assertLessEqual_ULINT : BOOL (* Returns TRUE if act <= xp. *)(* https://github.com/tkucic/iecUnitTest/blob/main/docs/docs/ns/Global/fc/assertLessEqual_ULINT.md *)
    VAR_INPUT
        act : ULINT; (*Variable to test*)
        xp : ULINT; (*Variable to test against*)
    END_VAR
END_FUNCTION
FUNCTION assertLessEqual_REAL : BOOL (* Returns TRUE if act <= xp. *)(* https://github.com/tkucic/iecUnitTest/blob/main/docs/docs/ns/Global/fc/assertLessEqual_REAL.md *)
    VAR_INPUT
        act : REAL; (*Variable to test*)
        xp : REAL; (*Variable to test against*)
    END_VAR
END_FUNCTION
FUNCTION assertLessEqual_LREAL : BOOL (* Returns TRUE if act <= xp. *)(* https://github.com/tkucic/iecUnitTest/blob/main/docs/docs/ns/Global/fc/assertLessEqual_LREAL.md *)
    VAR_INPUT
        act : LREAL; (*Variable to test*)
        xp : LREAL; (*Variable to test against*)
    END_VAR
END_FUNCTION
FUNCTION assertLessEqual_TIME : BOOL (* Returns TRUE if act <= xp. *)(* https://github.com/tkucic/iecUnitTest/blob/main/docs/docs/ns/Global/fc/assertLessEqual_TIME.md *)
    VAR_INPUT
        act : TIME; (*Variable to test*)
        xp : TIME; (*Variable to test against*)
    END_VAR
END_FUNCTION
FUNCTION assertLessEqual_LTIME : BOOL (* Returns TRUE if act <= xp. *)(* https://github.com/tkucic/iecUnitTest/blob/main/docs/docs/ns/Global/fc/assertLessEqual_LTIME.md *)
    VAR_INPUT
        act : LTIME; (*Variable to test*)
        xp : LTIME; (*Variable to test against*)
    END_VAR
END_FUNCTION
FUNCTION assertLessEqual_DATE : BOOL (* Returns TRUE if act <= xp. *)(* https://github.com/tkucic/iecUnitTest/blob/main/docs/docs/ns/Global/fc/assertLessEqual_DATE.md *)
    VAR_INPUT
        act : DATE; (*Variable to test*)
        xp : DATE; (*Variable to test against*)
    END_VAR
END_FUNCTION
FUNCTION assertLessEqual_LDATE : BOOL (* Returns TRUE if act <= xp. *)(* https://github.com/tkucic/iecUnitTest/blob/main/docs/docs/ns/Global/fc/assertLessEqual_LDATE.md *)
    VAR_INPUT
        act : LDATE; (*Variable to test*)
        xp : LDATE; (*Variable to test against*)
    END_VAR
END_FUNCTION
FUNCTION assertLessEqual_DATE_AND_TIME : BOOL (* Returns TRUE if act <= xp. *)(* https://github.com/tkucic/iecUnitTest/blob/main/docs/docs/ns/Global/fc/assertLessEqual_DATE_AND_TIME.md *)
    VAR_INPUT
        act : DT; (*Variable to test*)
        xp : DT; (*Variable to test against*)
    END_VAR
END_FUNCTION
FUNCTION assertLessEqual_LDATE_AND_TIME : BOOL (* Returns TRUE if act <= xp. *)(* https://github.com/tkucic/iecUnitTest/blob/main/docs/docs/ns/Global/fc/assertLessEqual_LDATE_AND_TIME.md *)
    VAR_INPUT
        act : LDATE_AND_TIME; (*Variable to test*)
        xp : LDATE_AND_TIME; (*Variable to test against*)
    END_VAR
END_FUNCTION
FUNCTION assertLessEqual_TIME_OF_DAY : BOOL (* Returns TRUE if act <= xp. *)(* https://github.com/tkucic/iecUnitTest/blob/main/docs/docs/ns/Global/fc/assertLessEqual_TIME_OF_DAY.md *)
    VAR_INPUT
        act : TOD; (*Variable to test*)
        xp : TOD; (*Variable to test against*)
    END_VAR
END_FUNCTION
FUNCTION assertLessEqual_LTIME_OF_DAY : BOOL (* Returns TRUE if act <= xp. *)(* https://github.com/tkucic/iecUnitTest/blob/main/docs/docs/ns/Global/fc/assertLessEqual_LTIME_OF_DAY.md *)
    VAR_INPUT
        act : LTIME_OF_DAY; (*Variable to test*)
        xp : LTIME_OF_DAY; (*Variable to test against*)
    END_VAR
END_FUNCTION
FUNCTION assertArrayEqual_BOOL : BOOL (* Returns TRUE if act == xp. *)(* https://github.com/tkucic/iecUnitTest/blob/main/docs/docs/ns/Global/fc/assertArrayEqual_BOOL.md *)
    VAR_INPUT
        act : POINTER TO ARRAY[0..32000] OF BOOL; (*Variable to test*)
        xp : POINTER TO ARRAY[0..32000] OF BOOL; (*Variable to test against*)
        size : UINT; (*Size of the array (ADR(act))*)
    END_VAR
    VAR
        i : UINT; (*Iterator variable*)
        vStop : UINT; (*Size of the array / End of iteration*)
        pt1 : POINTER TO BOOL; (*Pointer to the element of the array act*)
        pt2 : POINTER TO BOOL; (*Pointer to the element of the array xp*)
    END_VAR
END_FUNCTION
FUNCTION assertArrayEqual_BYTE : BOOL (* Returns TRUE if act == xp. *)(* https://github.com/tkucic/iecUnitTest/blob/main/docs/docs/ns/Global/fc/assertArrayEqual_BYTE.md *)
    VAR_INPUT
        act : POINTER TO ARRAY[0..32000] OF BYTE; (*Variable to test*)
        xp : POINTER TO ARRAY[0..32000] OF BYTE; (*Variable to test against*)
        size : UINT; (*Size of the array (ADR(act))*)
    END_VAR
    VAR
        i : UINT; (*Iterator variable*)
        vStop : UINT; (*Size of the array / End of iteration*)
        pt1 : POINTER TO BYTE; (*Pointer to the element of the array act*)
        pt2 : POINTER TO BYTE; (*Pointer to the element of the array xp*)
    END_VAR
END_FUNCTION
FUNCTION assertArrayEqual_WORD : BOOL (* Returns TRUE if act == xp. *)(* https://github.com/tkucic/iecUnitTest/blob/main/docs/docs/ns/Global/fc/assertArrayEqual_WORD.md *)
    VAR_INPUT
        act : POINTER TO ARRAY[0..32000] OF WORD; (*Variable to test*)
        xp : POINTER TO ARRAY[0..32000] OF WORD; (*Variable to test against*)
        size : UINT; (*Size of the array (ADR(act))*)
    END_VAR
    VAR
        i : UINT; (*Iterator variable*)
        vStop : UINT; (*Size of the array / End of iteration*)
        pt1 : POINTER TO WORD; (*Pointer to the element of the array act*)
        pt2 : POINTER TO WORD; (*Pointer to the element of the array xp*)
    END_VAR
END_FUNCTION
FUNCTION assertArrayEqual_DWORD : BOOL (* Returns TRUE if act == xp. *)(* https://github.com/tkucic/iecUnitTest/blob/main/docs/docs/ns/Global/fc/assertArrayEqual_DWORD.md *)
    VAR_INPUT
        act : POINTER TO ARRAY[0..32000] OF DWORD; (*Variable to test*)
        xp : POINTER TO ARRAY[0..32000] OF DWORD; (*Variable to test against*)
        size : UINT; (*Size of the array (ADR(act))*)
    END_VAR
    VAR
        i : UINT; (*Iterator variable*)
        vStop : UINT; (*Size of the array / End of iteration*)
        pt1 : POINTER TO DWORD; (*Pointer to the element of the array act*)
        pt2 : POINTER TO DWORD; (*Pointer to the element of the array xp*)
    END_VAR
END_FUNCTION
FUNCTION assertArrayEqual_LWORD : BOOL (* Returns TRUE if act == xp. *)(* https://github.com/tkucic/iecUnitTest/blob/main/docs/docs/ns/Global/fc/assertArrayEqual_LWORD.md *)
    VAR_INPUT
        act : POINTER TO ARRAY[0..32000] OF LWORD; (*Variable to test*)
        xp : POINTER TO ARRAY[0..32000] OF LWORD; (*Variable to test against*)
        size : UINT; (*Size of the array (ADR(act))*)
    END_VAR
    VAR
        i : UINT; (*Iterator variable*)
        vStop : UINT; (*Size of the array / End of iteration*)
        pt1 : POINTER TO LWORD; (*Pointer to the element of the array act*)
        pt2 : POINTER TO LWORD; (*Pointer to the element of the array xp*)
    END_VAR
END_FUNCTION
FUNCTION assertArrayEqual_SINT : BOOL (* Returns TRUE if act == xp. *)(* https://github.com/tkucic/iecUnitTest/blob/main/docs/docs/ns/Global/fc/assertArrayEqual_SINT.md *)
    VAR_INPUT
        act : POINTER TO ARRAY[0..32000] OF SINT; (*Variable to test*)
        xp : POINTER TO ARRAY[0..32000] OF SINT; (*Variable to test against*)
        size : UINT; (*Size of the array (ADR(act))*)
    END_VAR
    VAR
        i : UINT; (*Iterator variable*)
        vStop : UINT; (*Size of the array / End of iteration*)
        pt1 : POINTER TO SINT; (*Pointer to the element of the array act*)
        pt2 : POINTER TO SINT; (*Pointer to the element of the array xp*)
    END_VAR
END_FUNCTION
FUNCTION assertArrayEqual_USINT : BOOL (* Returns TRUE if act == xp. *)(* https://github.com/tkucic/iecUnitTest/blob/main/docs/docs/ns/Global/fc/assertArrayEqual_USINT.md *)
    VAR_INPUT
        act : POINTER TO ARRAY[0..32000] OF USINT; (*Variable to test*)
        xp : POINTER TO ARRAY[0..32000] OF USINT; (*Variable to test against*)
        size : UINT; (*Size of the array (ADR(act))*)
    END_VAR
    VAR
        i : UINT; (*Iterator variable*)
        vStop : UINT; (*Size of the array / End of iteration*)
        pt1 : POINTER TO USINT; (*Pointer to the element of the array act*)
        pt2 : POINTER TO USINT; (*Pointer to the element of the array xp*)
    END_VAR
END_FUNCTION
FUNCTION assertArrayEqual_INT : BOOL (* Returns TRUE if act == xp. *)(* https://github.com/tkucic/iecUnitTest/blob/main/docs/docs/ns/Global/fc/assertArrayEqual_INT.md *)
    VAR_INPUT
        act : POINTER TO ARRAY[0..32000] OF INT; (*Variable to test*)
        xp : POINTER TO ARRAY[0..32000] OF INT; (*Variable to test against*)
        size : UINT; (*Size of the array (ADR(act))*)
    END_VAR
    VAR
        i : UINT; (*Iterator variable*)
        vStop : UINT; (*Size of the array / End of iteration*)
        pt1 : POINTER TO INT; (*Pointer to the element of the array act*)
        pt2 : POINTER TO INT; (*Pointer to the element of the array xp*)
    END_VAR
END_FUNCTION
FUNCTION assertArrayEqual_UINT : BOOL (* Returns TRUE if act == xp. *)(* https://github.com/tkucic/iecUnitTest/blob/main/docs/docs/ns/Global/fc/assertArrayEqual_UINT.md *)
    VAR_INPUT
        act : POINTER TO ARRAY[0..32000] OF UINT; (*Variable to test*)
        xp : POINTER TO ARRAY[0..32000] OF UINT; (*Variable to test against*)
        size : UINT; (*Size of the array (ADR(act))*)
    END_VAR
    VAR
        i : UINT; (*Iterator variable*)
        vStop : UINT; (*Size of the array / End of iteration*)
        pt1 : POINTER TO UINT; (*Pointer to the element of the array act*)
        pt2 : POINTER TO UINT; (*Pointer to the element of the array xp*)
    END_VAR
END_FUNCTION
FUNCTION assertArrayEqual_DINT : BOOL (* Returns TRUE if act == xp. *)(* https://github.com/tkucic/iecUnitTest/blob/main/docs/docs/ns/Global/fc/assertArrayEqual_DINT.md *)
    VAR_INPUT
        act : POINTER TO ARRAY[0..32000] OF DINT; (*Variable to test*)
        xp : POINTER TO ARRAY[0..32000] OF DINT; (*Variable to test against*)
        size : UINT; (*Size of the array (ADR(act))*)
    END_VAR
    VAR
        i : UINT; (*Iterator variable*)
        vStop : UINT; (*Size of the array / End of iteration*)
        pt1 : POINTER TO DINT; (*Pointer to the element of the array act*)
        pt2 : POINTER TO DINT; (*Pointer to the element of the array xp*)
    END_VAR
END_FUNCTION
FUNCTION assertArrayEqual_UDINT : BOOL (* Returns TRUE if act == xp. *)(* https://github.com/tkucic/iecUnitTest/blob/main/docs/docs/ns/Global/fc/assertArrayEqual_UDINT.md *)
    VAR_INPUT
        act : POINTER TO ARRAY[0..32000] OF UDINT; (*Variable to test*)
        xp : POINTER TO ARRAY[0..32000] OF UDINT; (*Variable to test against*)
        size : UINT; (*Size of the array (ADR(act))*)
    END_VAR
    VAR
        i : UINT; (*Iterator variable*)
        vStop : UINT; (*Size of the array / End of iteration*)
        pt1 : POINTER TO UDINT; (*Pointer to the element of the array act*)
        pt2 : POINTER TO UDINT; (*Pointer to the element of the array xp*)
    END_VAR
END_FUNCTION
FUNCTION assertArrayEqual_LINT : BOOL (* Returns TRUE if act == xp. *)(* https://github.com/tkucic/iecUnitTest/blob/main/docs/docs/ns/Global/fc/assertArrayEqual_LINT.md *)
    VAR_INPUT
        act : POINTER TO ARRAY[0..32000] OF LINT; (*Variable to test*)
        xp : POINTER TO ARRAY[0..32000] OF LINT; (*Variable to test against*)
        size : UINT; (*Size of the array (ADR(act))*)
    END_VAR
    VAR
        i : UINT; (*Iterator variable*)
        vStop : UINT; (*Size of the array / End of iteration*)
        pt1 : POINTER TO LINT; (*Pointer to the element of the array act*)
        pt2 : POINTER TO LINT; (*Pointer to the element of the array xp*)
    END_VAR
END_FUNCTION
FUNCTION assertArrayEqual_ULINT : BOOL (* Returns TRUE if act == xp. *)(* https://github.com/tkucic/iecUnitTest/blob/main/docs/docs/ns/Global/fc/assertArrayEqual_ULINT.md *)
    VAR_INPUT
        act : POINTER TO ARRAY[0..32000] OF ULINT; (*Variable to test*)
        xp : POINTER TO ARRAY[0..32000] OF ULINT; (*Variable to test against*)
        size : UINT; (*Size of the array (ADR(act))*)
    END_VAR
    VAR
        i : UINT; (*Iterator variable*)
        vStop : UINT; (*Size of the array / End of iteration*)
        pt1 : POINTER TO ULINT; (*Pointer to the element of the array act*)
        pt2 : POINTER TO ULINT; (*Pointer to the element of the array xp*)
    END_VAR
END_FUNCTION
FUNCTION assertArrayEqual_REAL : BOOL (* Returns TRUE if act == xp. *)(* https://github.com/tkucic/iecUnitTest/blob/main/docs/docs/ns/Global/fc/assertArrayEqual_REAL.md *)
    VAR_INPUT
        act : POINTER TO ARRAY[0..32000] OF REAL; (*Variable to test*)
        xp : POINTER TO ARRAY[0..32000] OF REAL; (*Variable to test against*)
        size : UINT; (*Size of the array (ADR(act))*)
    END_VAR
    VAR
        i : UINT; (*Iterator variable*)
        vStop : UINT; (*Size of the array / End of iteration*)
        pt1 : POINTER TO REAL; (*Pointer to the element of the array act*)
        pt2 : POINTER TO REAL; (*Pointer to the element of the array xp*)
    END_VAR
END_FUNCTION
FUNCTION assertArrayEqual_LREAL : BOOL (* Returns TRUE if act == xp. *)(* https://github.com/tkucic/iecUnitTest/blob/main/docs/docs/ns/Global/fc/assertArrayEqual_LREAL.md *)
    VAR_INPUT
        act : POINTER TO ARRAY[0..32000] OF LREAL; (*Variable to test*)
        xp : POINTER TO ARRAY[0..32000] OF LREAL; (*Variable to test against*)
        size : UINT; (*Size of the array (ADR(act))*)
    END_VAR
    VAR
        i : UINT; (*Iterator variable*)
        vStop : UINT; (*Size of the array / End of iteration*)
        pt1 : POINTER TO LREAL; (*Pointer to the element of the array act*)
        pt2 : POINTER TO LREAL; (*Pointer to the element of the array xp*)
    END_VAR
END_FUNCTION
FUNCTION assertArrayEqual_STRING : BOOL (* Returns TRUE if act == xp. *)(* https://github.com/tkucic/iecUnitTest/blob/main/docs/docs/ns/Global/fc/assertArrayEqual_STRING.md *)
    VAR_INPUT
        act : POINTER TO ARRAY[0..32000] OF STRING; (*Variable to test*)
        xp : POINTER TO ARRAY[0..32000] OF STRING; (*Variable to test against*)
        size : UINT; (*Size of the array (ADR(act))*)
    END_VAR
    VAR
        i : UINT; (*Iterator variable*)
        vStop : UINT; (*Size of the array / End of iteration*)
        pt1 : POINTER TO STRING; (*Pointer to the element of the array act*)
        pt2 : POINTER TO STRING; (*Pointer to the element of the array xp*)
    END_VAR
END_FUNCTION
FUNCTION assertArrayEqual_WSTRING : BOOL (* Returns TRUE if act == xp. *)(* https://github.com/tkucic/iecUnitTest/blob/main/docs/docs/ns/Global/fc/assertArrayEqual_WSTRING.md *)
    VAR_INPUT
        act : POINTER TO ARRAY[0..32000] OF wstring; (*Variable to test*)
        xp : POINTER TO ARRAY[0..32000] OF wstring; (*Variable to test against*)
        size : UINT; (*Size of the array (ADR(act))*)
    END_VAR
    VAR
        i : UINT; (*Iterator variable*)
        vStop : UINT; (*Size of the array / End of iteration*)
        pt1 : POINTER TO wstring; (*Pointer to the element of the array act*)
        pt2 : POINTER TO wstring; (*Pointer to the element of the array xp*)
    END_VAR
END_FUNCTION
FUNCTION assertArrayEqual_TIME : BOOL (* Returns TRUE if act == xp. *)(* https://github.com/tkucic/iecUnitTest/blob/main/docs/docs/ns/Global/fc/assertArrayEqual_TIME.md *)
    VAR_INPUT
        act : POINTER TO ARRAY[0..32000] OF TIME; (*Variable to test*)
        xp : POINTER TO ARRAY[0..32000] OF TIME; (*Variable to test against*)
        size : UINT; (*Size of the array (ADR(act))*)
    END_VAR
    VAR
        i : UINT; (*Iterator variable*)
        vStop : UINT; (*Size of the array / End of iteration*)
        pt1 : POINTER TO TIME; (*Pointer to the element of the array act*)
        pt2 : POINTER TO TIME; (*Pointer to the element of the array xp*)
    END_VAR
END_FUNCTION
FUNCTION assertArrayEqual_LTIME : BOOL (* Returns TRUE if act == xp. *)(* https://github.com/tkucic/iecUnitTest/blob/main/docs/docs/ns/Global/fc/assertArrayEqual_LTIME.md *)
    VAR_INPUT
        act : POINTER TO ARRAY[0..32000] OF LTIME; (*Variable to test*)
        xp : POINTER TO ARRAY[0..32000] OF LTIME; (*Variable to test against*)
        size : UINT; (*Size of the array (ADR(act))*)
    END_VAR
    VAR
        i : UINT; (*Iterator variable*)
        vStop : UINT; (*Size of the array / End of iteration*)
        pt1 : POINTER TO LTIME; (*Pointer to the element of the array act*)
        pt2 : POINTER TO LTIME; (*Pointer to the element of the array xp*)
    END_VAR
END_FUNCTION
FUNCTION assertArrayEqual_DATE : BOOL (* Returns TRUE if act == xp. *)(* https://github.com/tkucic/iecUnitTest/blob/main/docs/docs/ns/Global/fc/assertArrayEqual_DATE.md *)
    VAR_INPUT
        act : POINTER TO ARRAY[0..32000] OF DATE; (*Variable to test*)
        xp : POINTER TO ARRAY[0..32000] OF DATE; (*Variable to test against*)
        size : UINT; (*Size of the array (ADR(act))*)
    END_VAR
    VAR
        i : UINT; (*Iterator variable*)
        vStop : UINT; (*Size of the array / End of iteration*)
        pt1 : POINTER TO DATE; (*Pointer to the element of the array act*)
        pt2 : POINTER TO DATE; (*Pointer to the element of the array xp*)
    END_VAR
END_FUNCTION
FUNCTION assertArrayEqual_LDATE : BOOL (* Returns TRUE if act == xp. *)(* https://github.com/tkucic/iecUnitTest/blob/main/docs/docs/ns/Global/fc/assertArrayEqual_LDATE.md *)
    VAR_INPUT
        act : POINTER TO ARRAY[0..32000] OF LDATE; (*Variable to test*)
        xp : POINTER TO ARRAY[0..32000] OF LDATE; (*Variable to test against*)
        size : UINT; (*Size of the array (ADR(act))*)
    END_VAR
    VAR
        i : UINT; (*Iterator variable*)
        vStop : UINT; (*Size of the array / End of iteration*)
        pt1 : POINTER TO LDATE; (*Pointer to the element of the array act*)
        pt2 : POINTER TO LDATE; (*Pointer to the element of the array xp*)
    END_VAR
END_FUNCTION
FUNCTION assertArrayEqual_DATE_AND_TIME : BOOL (* Returns TRUE if act == xp. *)(* https://github.com/tkucic/iecUnitTest/blob/main/docs/docs/ns/Global/fc/assertArrayEqual_DATE_AND_TIME.md *)
    VAR_INPUT
        act : POINTER TO ARRAY[0..32000] OF DT; (*Variable to test*)
        xp : POINTER TO ARRAY[0..32000] OF DT; (*Variable to test against*)
        size : UINT; (*Size of the array (ADR(act))*)
    END_VAR
    VAR
        i : UINT; (*Iterator variable*)
        vStop : UINT; (*Size of the array / End of iteration*)
        pt1 : POINTER TO DT; (*Pointer to the element of the array act*)
        pt2 : POINTER TO DT; (*Pointer to the element of the array xp*)
    END_VAR
END_FUNCTION
FUNCTION assertArrayEqual_LDATE_AND_TIME : BOOL (* Returns TRUE if act == xp. *)(* https://github.com/tkucic/iecUnitTest/blob/main/docs/docs/ns/Global/fc/assertArrayEqual_LDATE_AND_TIME.md *)
    VAR_INPUT
        act : POINTER TO ARRAY[0..32000] OF LDATE_AND_TIME; (*Variable to test*)
        xp : POINTER TO ARRAY[0..32000] OF LDATE_AND_TIME; (*Variable to test against*)
        size : UINT; (*Size of the array (ADR(act))*)
    END_VAR
    VAR
        i : UINT; (*Iterator variable*)
        vStop : UINT; (*Size of the array / End of iteration*)
        pt1 : POINTER TO LDATE_AND_TIME; (*Pointer to the element of the array act*)
        pt2 : POINTER TO LDATE_AND_TIME; (*Pointer to the element of the array xp*)
    END_VAR
END_FUNCTION
FUNCTION assertArrayEqual_TIME_OF_DAY : BOOL (* Returns TRUE if act == xp. *)(* https://github.com/tkucic/iecUnitTest/blob/main/docs/docs/ns/Global/fc/assertArrayEqual_TIME_OF_DAY.md *)
    VAR_INPUT
        act : POINTER TO ARRAY[0..32000] OF TOD; (*Variable to test*)
        xp : POINTER TO ARRAY[0..32000] OF TOD; (*Variable to test against*)
        size : UINT; (*Size of the array (ADR(act))*)
    END_VAR
    VAR
        i : UINT; (*Iterator variable*)
        vStop : UINT; (*Size of the array / End of iteration*)
        pt1 : POINTER TO TOD; (*Pointer to the element of the array act*)
        pt2 : POINTER TO TOD; (*Pointer to the element of the array xp*)
    END_VAR
END_FUNCTION
FUNCTION assertArrayEqual_LTIME_OF_DAY : BOOL (* Returns TRUE if act == xp. *)(* https://github.com/tkucic/iecUnitTest/blob/main/docs/docs/ns/Global/fc/assertArrayEqual_LTIME_OF_DAY.md *)
    VAR_INPUT
        act : POINTER TO ARRAY[0..32000] OF LTIME_OF_DAY; (*Variable to test*)
        xp : POINTER TO ARRAY[0..32000] OF LTIME_OF_DAY; (*Variable to test against*)
        size : UINT; (*Size of the array (ADR(act))*)
    END_VAR
    VAR
        i : UINT; (*Iterator variable*)
        vStop : UINT; (*Size of the array / End of iteration*)
        pt1 : POINTER TO LTIME_OF_DAY; (*Pointer to the element of the array act*)
        pt2 : POINTER TO LTIME_OF_DAY; (*Pointer to the element of the array xp*)
    END_VAR
END_FUNCTION
FUNCTION assertTrue : BOOL (* Returns TRUE if condition is TRUE *)(* https://github.com/tkucic/iecUnitTest/blob/main/docs/docs/ns/Global/fc/assertTrue.md *)
    VAR_INPUT
        condition : BOOL; (*Variable to test*)
    END_VAR
END_FUNCTION

(* ---- utTestReporter.st ---- *)
FUNCTION_BLOCK utTestReporter
    (*https://github.com/tkucic/iecUnitTest/blob/main/docs/docs/ns/Global/fb/utTestReporter.md*)
    (*Reset totals*)
    NrPousUnderTest := 0;
    NrOfTests := 0;
    NrTestsPassed := 0;
    NrTestsFailed := 0;
    PassRate := 0;
    TestsInProgress := FALSE;
    Error := FALSE;

    (*Count totals*)
    FOR i:=0 TO 500 DO
    	IF Results[i].Id > 0 THEN
    		(*Count existing POUs under test*)
    		NrPousUnderTest := NrPousUnderTest + 1;
    		(*Count the pass rate. Needs to be divided in the end by the number of total tests*)
    		PassRate := PassRate + Results[i].PassRate;
    		(*Count the number of tests*)
    		NrOfTests := NrOfTests + Results[i].TotalTests;
    		(*Count the number of tests passed*)
    		NrTestsPassed := NrTestsPassed + Results[i].TestsPassed;
    		(*Count the number of tests failed*)
    		NrTestsFailed := NrTestsFailed + Results[i].TestsFailed;

    		(*Indicators*)
    		IF Results[i].TestsRunning THEN
    			TestsInProgress := TRUE;
    		END_IF
    		IF Results[i].Error <> utErrors.NO_ERROR THEN
    			Error := TRUE;
    		END_IF
    	END_IF
    END_FOR
    PassRate := PassRate / NrPousUnderTest;
END_FUNCTION_BLOCK

(* ---- utTestSuite.st ---- *)
FUNCTION_BLOCK utTestSuite
    (*https://github.com/tkucic/iecUnitTest/blob/main/docs/docs/ns/Global/fb/utTestSuite.md*)
    (*Copy name of object under test*)
    Summary.Id := Id;
    Summary.Name := Name;

    (*Handle commands to start*)
    runCmd(CLK:=RunTests);
    resetCmd(CLK:=ResetTests);

    (*Calculate total number of tests and other flags*)
    Summary.TotalTests := 0;
    Summary.TestsPassed := 0;
    Summary.TestsFailed := 0;
    Summary.TestsRunning := FALSE;
    FOR i:=0 TO 20 DO
    	IF TestCases[i].id > 0 THEN
    		Summary.TotalTests := Summary.TotalTests + 1;
    	END_IF
    	(*Start the test if the Run command is true, the test exists and it is in setup state*)
    	IF TestCases[i].id > 0 AND TestCases[i].state = utTestCaseStates.SETUP AND runCmd.Q THEN
    		TestCases[i].state := utTestCaseStates.RUNNING;
    	END_IF

    	(*Reset the test if the test exists and its PASSED or FAILED*)
    	IF TestCases[i].id > 0 AND TestCases[i].state > utTestCaseStates.RUNNING AND resetCmd.Q THEN
    		TestCases[i].state := utTestCaseStates.SETUP;
    	END_IF

    	(*Check the states of the test cases*)
    	IF TestCases[i].state = utTestCaseStates.RUNNING THEN
    		Summary.TestsRunning := TRUE;
    	END_IF
    	IF TestCases[i].state = utTestCaseStates.PASSED THEN
    		Summary.TestsPassed := Summary.TestsPassed + 1;
    	END_IF
    	IF TestCases[i].state = utTestCaseStates.FAILED THEN
    		Summary.TestsFailed := Summary.TestsFailed + 1;
    	END_IF
    END_FOR

    (*Error if number of tests defined is 0*)
    IF Summary.TotalTests = 0 THEN
    	Summary.Error := utErrors.NO_TEST_CASES_DEFINED;
    	RETURN;
    END_IF

    (*Calculate the pass rate if all tests have finished*)
    IF NOT Summary.TestsRunning THEN
    	Summary.PassRate := (Summary.TestsPassed / UINT_TO_REAL(Summary.TotalTests)) * 100.0;
    ELSE
    	Summary.PassRate := 0;
    END_IF
END_FUNCTION_BLOCK
